short summary
=================
This assertion method checks if the current string ``stringToCheck`` length
is equal to ``expectedLength``

.. <legal notes>

legal notes
=================
| SPDX-FileCopyrightText: © 2022 ekvip automation GmbH <info@ekvip.de>
| SPDX-License-Identifier: Apache-2.0
| For details check: Apache-2.0_

.. _Apache-2.0: https://www.apache.org/licenses/LICENSE-2.0

.. </legal notes>

parameters
=================

*)

METHOD lenghtIsExact
VAR_INPUT
	(* current string to check *)
	stringToCheck	:WSTRING(Tc2_System.MAX_STRING_LENGTH);
	(* expected length of ``stringToCheck`` *)
	expectedLength	:USINT;
	(* message if the assertion is false *)
	message			:AssertMessage;
END_VAR
END_METHOD

(*

short summary
=================
This assertion method checks if the current string ``stringToCheck`` length
is equal or less than to ``maxLength``

.. <legal notes>

legal notes
=================
| SPDX-FileCopyrightText: © 2022 ekvip automation GmbH <info@ekvip.de>
| SPDX-License-Identifier: Apache-2.0
| For details check: Apache-2.0_

.. _Apache-2.0: https://www.apache.org/licenses/LICENSE-2.0

.. </legal notes>

parameters
=================

*)

METHOD lenghtIsMax
VAR_INPUT
	(* current string to check *)
	stringToCheck	:WSTRING(Tc2_System.MAX_STRING_LENGTH);
	(* upper limit of the length of ``stringToCheck`` *)
	maxLength		:USINT;
	(* message if the assertion is false *)
	message			:AssertMessage;
END_VAR
END_METHOD

(*

short summary
=================
This assertion method checks if the current string ``stringToCheck`` length
is equal or grater than to ``minLength``

.. <legal notes>

legal notes
=================
| SPDX-FileCopyrightText: © 2022 ekvip automation GmbH <info@ekvip.de>
| SPDX-License-Identifier: Apache-2.0
| For details check: Apache-2.0_

.. _Apache-2.0: https://www.apache.org/licenses/LICENSE-2.0

.. </legal notes>

parameters
=================

*)

METHOD lenghtIsMin
VAR_INPUT
	(* current string to check *)
	stringToCheck	:WSTRING(Tc2_System.MAX_STRING_LENGTH);
	(* lower limit of the length of ``stringToCheck`` *)
	minLength	:USINT;
	(* message if the assertion is false *)
	message			:AssertMessage;
END_VAR
END_METHOD

(*

short summary
=================
This assertion method checks if the current string ``stringToCheck`` starts with ``start``

.. attention:: 
	start of the string is **ALWAYS** the left side of the string 
	even for writings which written from right to left like Hebrew or Arabic

.. <legal notes>

legal notes
=================
| SPDX-FileCopyrightText: © 2022 ekvip automation GmbH <info@ekvip.de>
| SPDX-License-Identifier: Apache-2.0
| For details check: Apache-2.0_

.. _Apache-2.0: https://www.apache.org/licenses/LICENSE-2.0

.. </legal notes>

parameters
=================

*)

METHOD startsWith
VAR_INPUT
	(* current string to check *)
	stringToCheck	:WSTRING(Tc2_System.MAX_STRING_LENGTH);
	(* expected start of ``stringToCheck`` *)
	start			:WSTRING(Tc2_System.MAX_STRING_LENGTH);
	(* ``TRUE`` means ignore cases; ``FALSE`` means cases must be equal too *)
	ignoreCases		:BOOL;
	(* ``TRUE`` means truncation of spaces on the left side of ``stringToCheck``*)
	trim			:BOOL;
	(* message if the assertion is false *)
	message			:AssertMessage;
END_VAR
END_METHOD

END_INTERFACE

// ---- Assertor/Assertions/StringAssertion/WString/interfaces/IUtf16StringPointerAssertions.TcIO
(*

short summary
=================
This interface provides assert statements for UTF-16 strings

.. attention:: 
	All strings are handled as null terminated word streams.
	For UTF-16 is end of the string 16#00_00

.. <legal notes>

legal notes
=================
| SPDX-FileCopyrightText: © 2022 ekvip automation GmbH <info@ekvip.de>
| SPDX-License-Identifier: Apache-2.0
| For details check: Apache-2.0_

.. _Apache-2.0: https://www.apache.org/licenses/LICENSE-2.0

.. </legal notes>

methods
==================

*)

INTERFACE IUtf16StringPointerAssertions EXTENDS IAssertCallBackSetter

(*

short summary
=================
This assertion method for UTF-16 strings checks if the current string ``stringToCheck`` contains the search string ``searchString``

.. attention:: 
	All strings are handled as null terminated word streams.
	For UTF-16 is end of the string 16#00_00

.. <legal notes>

legal notes
=================
| SPDX-FileCopyrightText: © 2022 ekvip automation GmbH <info@ekvip.de>
| SPDX-License-Identifier: Apache-2.0
| For details check: Apache-2.0_

.. _Apache-2.0: https://www.apache.org/licenses/LICENSE-2.0

.. </legal notes>

parameters
=================

*)

METHOD utf16Contains
VAR_INPUT
	(* current string to check *)
	stringToCheck	:POINTER TO WORD;
	(* string must be found in ``stringToCheck`` *)
	searchString	:POINTER TO WORD;
	(* ``TRUE`` means ignore cases; ``FALSE`` means cases must be equal too *)
	ignoreCases		:BOOL;
	(* message if the assertion is false *)
	message			:AssertMessage;
END_VAR
END_METHOD

(*

short summary
=================
This assertion method for UTF-16 strings checks if the current string ``stringToCheck`` contains not the search string ``searchString``

.. attention:: 
	All strings are handled as null terminated word streams.
	For UTF-16 is end of the string 16#00_00

.. <legal notes>

legal notes
=================
| SPDX-FileCopyrightText: © 2022 ekvip automation GmbH <info@ekvip.de>
| SPDX-License-Identifier: Apache-2.0
| For details check: Apache-2.0_

.. _Apache-2.0: https://www.apache.org/licenses/LICENSE-2.0

.. </legal notes>

parameters
=================

*)

METHOD utf16ContainsNo
VAR_INPUT
	(* current string to check *)
	stringToCheck	:POINTER TO WORD;
	(* string must be found in ``stringToCheck`` *)
	searchString	:POINTER TO WORD;
	(* ``TRUE`` means ignore cases; ``FALSE`` means cases must be equal too *)
	ignoreCases		:BOOL;
	(* message if the assertion is false *)
	message			:AssertMessage;
END_VAR
END_METHOD

(*

short summary
=================
This assertion method for UTF-16 strings checks if the current string ``stringToCheck`` ends with the string ``end``

.. attention:: 
	All strings are handled as null terminated word streams.
	For UTF-16 is end of the string 16#00_00

.. attention:: 
	end of the string is **ALWAYS** the right side of the string 
	even for writings which written from right to left like Hebrew or Arabic

.. <legal notes>

legal notes
=================
| SPDX-FileCopyrightText: © 2022 ekvip automation GmbH <info@ekvip.de>
| SPDX-License-Identifier: Apache-2.0
| For details check: Apache-2.0_

.. _Apache-2.0: https://www.apache.org/licenses/LICENSE-2.0

.. </legal notes>

parameters
=================

*)

METHOD utf16EndsWith
VAR_INPUT
	(* current string to check *)
	stringToCheck	:POINTER TO WORD;
	(* string must be the end of ``stringToCheck`` *)
	end				:POINTER TO WORD;
	(* ``TRUE`` means ignore cases; ``FALSE`` means cases must be equal too *)
	ignoreCases		:BOOL;
	(* ``TRUE`` means truncation of spaces on the right side of ``stringToCheck``*)
	trim			:BOOL;
	(* message if the assertion is false *)
	message			:AssertMessage;
END_VAR
END_METHOD

(*

short summary
=================
This assertion method for utf-16 strings checks if the current string ``stringToCheck`` is equal to the ``expected`` string

.. attention:: 
	All strings are handled as null terminated word streams.
	For UTF-16 is end of the string 16#00_00

.. <legal notes>

legal notes
=================
| SPDX-FileCopyrightText: © 2022 ekvip automation GmbH <info@ekvip.de>
| SPDX-License-Identifier: Apache-2.0
| For details check: Apache-2.0_

.. _Apache-2.0: https://www.apache.org/licenses/LICENSE-2.0

.. </legal notes>

parameters
=================

*)

METHOD utf16IsEqualTo
VAR_INPUT
	(* current string to check *)
	stringToCheck	:POINTER TO WORD;
	(* ``stringToCheck`` must be equal to expected *)
	expected		:POINTER TO WORD;
	(* ``TRUE`` means ignore cases; ``FALSE`` means cases must be equal too *)
	ignoreCases		:BOOL;
	(* message if the assertion is false *)
	message			:AssertMessage;
END_VAR
END_METHOD

(*

short summary
=================
This assertion method for utf-16 strings checks if the current string ``stringToCheck`` is not equal to the ``unexpected`` string

.. attention:: 
	All strings are handled as null terminated word streams.
	For UTF-16 is end of the string 16#00_00

.. <legal notes>

legal notes
=================
| SPDX-FileCopyrightText: © 2022 ekvip automation GmbH <info@ekvip.de>
| SPDX-License-Identifier: Apache-2.0
| For details check: Apache-2.0_

.. _Apache-2.0: https://www.apache.org/licenses/LICENSE-2.0

.. </legal notes>

parameters
=================

*)

METHOD utf16IsNotEqualTo
VAR_INPUT
	(* current string to check *)
	stringToCheck	:POINTER TO WORD;
	(* ``stringToCheck`` must be not equal to unexpected *)
	unexpected		:POINTER TO WORD;
	(* ``TRUE`` means ignore cases; ``FALSE`` means cases must be equal too *)
	ignoreCases		:BOOL;
	(* message if the assertion is false *)
	message			:AssertMessage;
END_VAR
END_METHOD

(*

short summary
=================
This assertion method checks if the current string ``stringToCheck`` is length
is equal to ``expectedLength``

.. attention:: 
	All strings are handled as null terminated word streams.
	For UTF-16 is end of the string 16#00_00

.. <legal notes>

legal notes
=================
| SPDX-FileCopyrightText: © 2022 ekvip automation GmbH <info@ekvip.de>
| SPDX-License-Identifier: Apache-2.0
| For details check: Apache-2.0_

.. _Apache-2.0: https://www.apache.org/licenses/LICENSE-2.0

.. </legal notes>

parameters
=================

*)

METHOD utf16LenghtIsExact
VAR_INPUT
	(* current string to check *)
	stringToCheck	:POINTER TO WORD;
	(* expected length of ``stringToCheck`` *)
	expectedLength	:UDINT;
	(* message if the assertion is false *)
	message			:AssertMessage;
END_VAR
END_METHOD

(*

short summary
=================
This assertion method checks if the current string ``stringToCheck`` is length
is equal or less than to ``maxLength``

.. attention:: 
	All strings are handled as null terminated word streams.
	For UTF-16 is end of the string 16#00_00

.. <legal notes>

legal notes
=================
| SPDX-FileCopyrightText: © 2022 ekvip automation GmbH <info@ekvip.de>
| SPDX-License-Identifier: Apache-2.0
| For details check: Apache-2.0_

.. _Apache-2.0: https://www.apache.org/licenses/LICENSE-2.0

.. </legal notes>

parameters
=================

*)

METHOD utf16LenghtIsMax
VAR_INPUT
	(* current string to check *)
	stringToCheck	:POINTER TO WORD;
	(* upper limit of the length of ``stringToCheck`` *)
	maxLength		:UDINT;
	(* message if the assertion is false *)
	message			:AssertMessage;
END_VAR
END_METHOD

(*

short summary
=================
This assertion method checks if the current string ``stringToCheck`` is length
is equal or grater than to ``minLength``

.. attention:: 
	All strings are handled as null terminated word streams.
	For UTF-16 is end of the string 16#00_00

.. <legal notes>

legal notes
=================
| SPDX-FileCopyrightText: © 2022 ekvip automation GmbH <info@ekvip.de>
| SPDX-License-Identifier: Apache-2.0
| For details check: Apache-2.0_

.. _Apache-2.0: https://www.apache.org/licenses/LICENSE-2.0

.. </legal notes>

parameters
=================

*)

METHOD utf16LenghtIsMin
VAR_INPUT
	(* current string to check *)
	stringToCheck	:POINTER TO WORD;
	(* lower limit of the length of ``stringToCheck`` *)
	minLength		:UDINT;
	(* message if the assertion is false *)
	message			:AssertMessage;
END_VAR
END_METHOD

(*

short summary
=================
This assertion method checks if the current string ``stringToCheck`` is length
is equal or grater than ``minLength`` and equal or less than ``maxLength``

.. attention:: 
	All strings are handled as null terminated word streams.
	For UTF-16 is end of the string 16#00_00

.. <legal notes>

legal notes
=================
| SPDX-FileCopyrightText: © 2022 ekvip automation GmbH <info@ekvip.de>
| SPDX-License-Identifier: Apache-2.0
| For details check: Apache-2.0_

.. _Apache-2.0: https://www.apache.org/licenses/LICENSE-2.0

.. </legal notes>

parameters
=================

*)

METHOD utf16LengthIsBetween
VAR_INPUT
	(* current string to check *)
	stringToCheck	:POINTER TO WORD;
	(* lower limit of the string length *)
	minLenght		:UDINT;
	(* upper limit of the string length *)
	maxLenght		:UDINT;
	(* message if the assertion is false *)
	message			:AssertMessage;
END_VAR
END_METHOD

(*

short summary
=================
This assertion method for UTF-16 strings checks if the current string ``stringToCheck`` strats with the string ``start``

.. attention:: 
	All strings are handled as null terminated word streams.
	For UTF-16 is end of the string 16#00_00

.. attention:: 
	start of the string is **ALWAYS** the left side of the string 
	even for writings which written from right to left like Hebrew or Arabic

.. <legal notes>

legal notes
=================
| SPDX-FileCopyrightText: © 2022 ekvip automation GmbH <info@ekvip.de>
| SPDX-License-Identifier: Apache-2.0
| For details check: Apache-2.0_

.. _Apache-2.0: https://www.apache.org/licenses/LICENSE-2.0

.. </legal notes>

parameters
=================

*)

METHOD utf16StartsWith
VAR_INPUT
	(* current string to check *)
	stringToCheck	:POINTER TO WORD;
	(* expected start of ``stringToCheck`` *)
	start			:POINTER TO WORD;
	(* ``TRUE`` means ignore cases; ``FALSE`` means cases must be equal too *)
	ignoreCases		:BOOL;
	(* ``TRUE`` means truncation of spaces on the right side of ``stringToCheck``*)
	trim			:BOOL;
	(* message if the assertion is false *)
	message			:AssertMessage;
END_VAR
END_METHOD

END_INTERFACE

// ---- Assertor/Assertions/TimeAssertions/interfaces/ITimeAssertions.TcIO
(*

short summary
=================
This interface provides assert statements for times
For ``LTIME`` assertions use the property :ref:`ITimeAssertions.long`.
For ``TIME`` assertions use the property :ref:`ITimeAssertions.simple`.
.. <legal notes>

legal notes
=================
| SPDX-FileCopyrightText: © 2022 ekvip automation GmbH <info@ekvip.de>
| SPDX-License-Identifier: Apache-2.0
| For details check: Apache-2.0_

.. _Apache-2.0: https://www.apache.org/licenses/LICENSE-2.0

.. </legal notes>

methods
==================

*)

INTERFACE ITimeAssertions EXTENDS __SYSTEM.IQueryInterface

(*

short summary
=================
Returns an interface with assert statements for 64 bit times 

.. <legal notes>

legal notes
=================
| SPDX-FileCopyrightText: © 2022 ekvip automation GmbH <info@ekvip.de>
| SPDX-License-Identifier: Apache-2.0
| For details check: Apache-2.0_

.. _Apache-2.0: https://www.apache.org/licenses/LICENSE-2.0

.. </legal notes>

*)

PROPERTY long :I64BitTimeAssertions
GET
END_GET
END_PROPERTY

(*

short summary
=================
Returns an interface with assert statements for 32 bit times 

.. <legal notes>

legal notes
=================
| SPDX-FileCopyrightText: © 2022 ekvip automation GmbH <info@ekvip.de>
| SPDX-License-Identifier: Apache-2.0
| For details check: Apache-2.0_

.. _Apache-2.0: https://www.apache.org/licenses/LICENSE-2.0

.. </legal notes>

*)

PROPERTY simple :I32BitTimeAssertions
GET
END_GET
END_PROPERTY

END_INTERFACE

// ---- Assertor/Assertions/TimeAssertions/LTime/interfaces/I64BitTimeAssertions.TcIO
(*

short summary
=================
This interface provides assert statements for 64 bit ``LTIME``  

.. <legal notes>

legal notes
=================
| SPDX-FileCopyrightText: © 2022 ekvip automation GmbH <info@ekvip.de>
| SPDX-License-Identifier: Apache-2.0
| For details check: Apache-2.0_

.. _Apache-2.0: https://www.apache.org/licenses/LICENSE-2.0

.. </legal notes>

methods
==================

*)

INTERFACE I64BitTimeAssertions EXTENDS __SYSTEM.IQueryInterface

(*

short summary
=================
This assertion method checks whether time has elapsed since the timestamp time

.. <legal notes>

legal notes
=================
| SPDX-FileCopyrightText: © 2022 ekvip automation GmbH <info@ekvip.de>
| SPDX-License-Identifier: Apache-2.0
| For details check: Apache-2.0_

.. _Apache-2.0: https://www.apache.org/licenses/LICENSE-2.0

.. </legal notes>

parameters
=================

*)

METHOD timeHasExpired
VAR_INPUT
	(* start time you get it with ``LTIME()`` *)
	timestamp		:LTIME;
	(* timeout like ``LTIME#300ms`` *)
	expiringTime	:LTIME;
	(* message if the assertion is false *)
	message			:AssertMessage;
END_VAR
END_METHOD

(*

short summary
=================
This assertion method checks that the time since the timestamp time has not yet elapsed

.. <legal notes>

legal notes
=================
| SPDX-FileCopyrightText: © 2022 ekvip automation GmbH <info@ekvip.de>
| SPDX-License-Identifier: Apache-2.0
| For details check: Apache-2.0_

.. _Apache-2.0: https://www.apache.org/licenses/LICENSE-2.0

.. </legal notes>

parameters
=================

*)

METHOD timeHasNotExpired
VAR_INPUT
	(* start time you get it with ``LTIME()`` *)
	timestamp		:LTIME;
	(* timeout like ``LTIME#300ms`` *)
	expiringTime	:LTIME;
	(* message if the assertion is false *)
	message			:AssertMessage;
END_VAR
END_METHOD

(*

short summary
=================
This assertion method checks if the current value is equal to the expected value

.. <legal notes>

legal notes
=================
| SPDX-FileCopyrightText: © 2022 ekvip automation GmbH <info@ekvip.de>
| SPDX-License-Identifier: Apache-2.0
| For details check: Apache-2.0_

.. _Apache-2.0: https://www.apache.org/licenses/LICENSE-2.0

.. </legal notes>

parameters
=================

*)

METHOD valueIsEqualTo
VAR_INPUT
	(* current value to check *)
	currentValue	:LTIME;
	(* expected value to compare *)
	expectedValue	:LTIME;
	(* message if the assertion is false *)
	message			:AssertMessage;
END_VAR
END_METHOD

(*

short summary
=================
This assertion method checks if the current value is greater than the less value

.. <legal notes>

legal notes
=================
| SPDX-FileCopyrightText: © 2022 ekvip automation GmbH <info@ekvip.de>
| SPDX-License-Identifier: Apache-2.0
| For details check: Apache-2.0_

.. _Apache-2.0: https://www.apache.org/licenses/LICENSE-2.0

.. </legal notes>

parameters
=================

*)

METHOD valueIsGreaterThan
VAR_INPUT
	(* current value to check *)
	currentValue	:LTIME;
	(* less than lower limit *)
	lessValue		:LTIME;
	(* message if the assertion is false *)
	message			:AssertMessage;
END_VAR
END_METHOD

(*

short summary
=================
This assertion method checks if the current value is inside a limit

.. attention:: 
	limits are included: ``valueIsInRangeOf(lt#3ms,lt#3ms ,lt#3ms)`` is a true assertion

.. <legal notes>

legal notes
=================
| SPDX-FileCopyrightText: © 2022 ekvip automation GmbH <info@ekvip.de>
| SPDX-License-Identifier: Apache-2.0
| For details check: Apache-2.0_

.. _Apache-2.0: https://www.apache.org/licenses/LICENSE-2.0

.. </legal notes>

parameters
=================

*)

METHOD valueIsInRangeOf
VAR_INPUT
	(* lower limit for the current value *)
	lowerLimit		:LTIME;
	(* current value to check *)
	currentValue	:LTIME;
	(* upper limit for the current value *)
	upperLimit		:LTIME;
	(* message if the assertion is false *)
	message			:AssertMessage;
END_VAR
END_METHOD

(*

short summary
=================
This assertion method checks if the current value is less than the greater value

.. <legal notes>

legal notes
=================
| SPDX-FileCopyrightText: © 2022 ekvip automation GmbH <info@ekvip.de>
| SPDX-License-Identifier: Apache-2.0
| For details check: Apache-2.0_

.. _Apache-2.0: https://www.apache.org/licenses/LICENSE-2.0

.. </legal notes>

parameters
=================

*)

METHOD valueIsLessThan
VAR_INPUT
	(* current value to check *)
	currentValue	:LTIME;
	(* greater than upper limit *)
	greaterValue	:LTIME;
	(* message if the assertion is false *)
	message			:AssertMessage;
END_VAR
END_METHOD

(*

short summary
=================
This assertion method checks if the current value is less than or equal to the maximum value

.. <legal notes>

legal notes
=================
| SPDX-FileCopyrightText: © 2022 ekvip automation GmbH <info@ekvip.de>
| SPDX-License-Identifier: Apache-2.0
| For details check: Apache-2.0_

.. _Apache-2.0: https://www.apache.org/licenses/LICENSE-2.0

.. </legal notes>

parameters
=================

*)

METHOD valueIsMax
VAR_INPUT
	(* current value to check *)
	currentValue	:LTIME;
	(* upper limit for the current value *)
	maximumValue	:LTIME;
	(* message if the assertion is false *)
	message			:AssertMessage;
END_VAR
END_METHOD

(*

short summary
=================
This assertion method checks if the current value is greater than or equal to the minimum value

.. <legal notes>

legal notes
=================
| SPDX-FileCopyrightText: © 2022 ekvip automation GmbH <info@ekvip.de>
| SPDX-License-Identifier: Apache-2.0
| For details check: Apache-2.0_

.. _Apache-2.0: https://www.apache.org/licenses/LICENSE-2.0

.. </legal notes>

parameters
=================

*)

METHOD valueIsMin
VAR_INPUT
	(* current value to check *)
	currentValue	:LTIME;
	(* lower limit for the current value *)
	minimumValue	:LTIME;
	(* message if the assertion is false *)
	message			:AssertMessage;
END_VAR
END_METHOD

(*

short summary
=================
This assertion method checks if the current value is not equal to the unexpected value

.. <legal notes>

legal notes
=================
| SPDX-FileCopyrightText: © 2022 ekvip automation GmbH <info@ekvip.de>
| SPDX-License-Identifier: Apache-2.0
| For details check: Apache-2.0_

.. _Apache-2.0: https://www.apache.org/licenses/LICENSE-2.0

.. </legal notes>

parameters
=================

*)

METHOD valueIsNotEqualTo
VAR_INPUT
	(* current value to check *)
	currentValue	:LTIME;
	(* unexpected value to compare *)
	unexpectedValue	:LTIME;
	(* message if the assertion is false *)
	message			:AssertMessage;
END_VAR
END_METHOD

END_INTERFACE

// ---- Assertor/Assertions/TimeAssertions/Time/interfaces/I32BitTimeAssertions.TcIO
(*

short summary
=================
This interface provides assert statements for 32 bit ``TIME``  

.. <legal notes>

legal notes
=================
| SPDX-FileCopyrightText: © 2022 ekvip automation GmbH <info@ekvip.de>
| SPDX-License-Identifier: Apache-2.0
| For details check: Apache-2.0_

.. _Apache-2.0: https://www.apache.org/licenses/LICENSE-2.0

.. </legal notes>

methods
==================

*)

INTERFACE I32BitTimeAssertions EXTENDS __SYSTEM.IQueryInterface

(*

short summary
=================
This assertion method checks whether time has elapsed since the timestamp time

.. <legal notes>

legal notes
=================
| SPDX-FileCopyrightText: © 2022 ekvip automation GmbH <info@ekvip.de>
| SPDX-License-Identifier: Apache-2.0
| For details check: Apache-2.0_

.. _Apache-2.0: https://www.apache.org/licenses/LICENSE-2.0

.. </legal notes>

parameters
=================

*)

METHOD timeHasExpired
VAR_INPUT
	(* start time you get it with ``TIME()`` *)
	timestamp		:TIME;
	(* timeout like ``t#300ms`` *)
	expiringTime	:TIME;
	(* message if the assertion is false *)
	message			:AssertMessage;
END_VAR
END_METHOD

(*

short summary
=================
This assertion method checks that the time since the timestamp time has not yet elapsed

.. <legal notes>

legal notes
=================
| SPDX-FileCopyrightText: © 2022 ekvip automation GmbH <info@ekvip.de>
| SPDX-License-Identifier: Apache-2.0
| For details check: Apache-2.0_

.. _Apache-2.0: https://www.apache.org/licenses/LICENSE-2.0

.. </legal notes>

parameters
=================

*)

METHOD timeHasNotExpired
VAR_INPUT
	(* start time you get it with ``TIME()`` *)
	timestamp		:TIME;
	(* timeout like ``t#300ms`` *)
	expiringTime	:TIME;
	(* message if the assertion is false *)
	message			:AssertMessage;
END_VAR
END_METHOD

(*

short summary
=================
This assertion method checks if the current value is equal to the expected value

.. <legal notes>

legal notes
=================
| SPDX-FileCopyrightText: © 2022 ekvip automation GmbH <info@ekvip.de>
| SPDX-License-Identifier: Apache-2.0
| For details check: Apache-2.0_

.. _Apache-2.0: https://www.apache.org/licenses/LICENSE-2.0

.. </legal notes>

parameters
=================

*)

METHOD valueIsEqualTo
VAR_INPUT
	(* current value to check *)
	currentValue	:TIME;
	(* expected value to compare *)
	expectedValue	:TIME;
	(* message if the assertion is false *)
	message			:AssertMessage;
END_VAR
END_METHOD

(*

short summary
=================
This assertion method checks if the current value is greater than the less value

.. <legal notes>

legal notes
=================
| SPDX-FileCopyrightText: © 2022 ekvip automation GmbH <info@ekvip.de>
| SPDX-License-Identifier: Apache-2.0
| For details check: Apache-2.0_

.. _Apache-2.0: https://www.apache.org/licenses/LICENSE-2.0

.. </legal notes>

parameters
=================

*)

METHOD valueIsGreaterThan
VAR_INPUT
	(* current value to check *)
	currentValue	:TIME;
	(* less than lower limit *)
	lessValue		:TIME;
	(* message if the assertion is false *)
	message			:AssertMessage;
END_VAR
END_METHOD

(*

short summary
=================
This assertion method checks if the current value is inside a limit

.. attention:: 
	limits are included: ``valueIsInRangeOf(t#3ms,t#3ms ,t#3ms)`` is a true assertion

.. <legal notes>

legal notes
=================
| SPDX-FileCopyrightText: © 2022 ekvip automation GmbH <info@ekvip.de>
| SPDX-License-Identifier: Apache-2.0
| For details check: Apache-2.0_

.. _Apache-2.0: https://www.apache.org/licenses/LICENSE-2.0

.. </legal notes>

parameters
=================

*)

METHOD valueIsInRangeOf
VAR_INPUT
	(* lower limit for the current value *)
	lowerLimit		:TIME;
	(* current value to check *)
	currentValue	:TIME;
	(* upper limit for the current value *)
	upperLimit		:TIME;
	(* message if the assertion is false *)
	message			:AssertMessage;
END_VAR
END_METHOD

(*

short summary
=================
This assertion method checks if the current value is less than the greater value

.. <legal notes>

legal notes
=================
| SPDX-FileCopyrightText: © 2022 ekvip automation GmbH <info@ekvip.de>
| SPDX-License-Identifier: Apache-2.0
| For details check: Apache-2.0_

.. _Apache-2.0: https://www.apache.org/licenses/LICENSE-2.0

.. </legal notes>

parameters
=================

*)

METHOD valueIsLessThan
VAR_INPUT
	(* current value to check *)
	currentValue	:TIME;
	(* greater than upper limit *)
	greaterValue	:TIME;
	(* message if the assertion is false *)
	message			:AssertMessage;
END_VAR
END_METHOD

(*

short summary
=================
This assertion method checks if the current value is less than or equal to the maximum value

.. <legal notes>

legal notes
=================
| SPDX-FileCopyrightText: © 2022 ekvip automation GmbH <info@ekvip.de>
| SPDX-License-Identifier: Apache-2.0
| For details check: Apache-2.0_

.. _Apache-2.0: https://www.apache.org/licenses/LICENSE-2.0

.. </legal notes>

parameters
=================

*)

METHOD valueIsMax
VAR_INPUT
	(* current value to check *)
	currentValue	:TIME;
	(* upper limit for the current value *)
	maximumValue	:TIME;
	(* message if the assertion is false *)
	message			:AssertMessage;
END_VAR
END_METHOD

(*

short summary
=================
This assertion method checks if the current value is greater than or equal to the minimum value

.. <legal notes>

legal notes
=================
| SPDX-FileCopyrightText: © 2022 ekvip automation GmbH <info@ekvip.de>
| SPDX-License-Identifier: Apache-2.0
| For details check: Apache-2.0_

.. _Apache-2.0: https://www.apache.org/licenses/LICENSE-2.0

.. </legal notes>

parameters
=================

*)

METHOD valueIsMin
VAR_INPUT
	(* current value to check *)
	currentValue	:TIME;
	(* lower limit for the current value *)
	minimumValue	:TIME;
	(* message if the assertion is false *)
	message			:AssertMessage;
END_VAR
END_METHOD

(*

short summary
=================
This assertion method checks if the current value is not equal to the unexpected value

.. <legal notes>

legal notes
=================
| SPDX-FileCopyrightText: © 2022 ekvip automation GmbH <info@ekvip.de>
| SPDX-License-Identifier: Apache-2.0
| For details check: Apache-2.0_

.. _Apache-2.0: https://www.apache.org/licenses/LICENSE-2.0

.. </legal notes>

parameters
=================

*)

METHOD valueIsNotEqualTo
VAR_INPUT
	(* current value to check *)
	currentValue	:TIME;
	(* unexpected value to compare *)
	unexpectedValue	:TIME;
	(* message if the assertion is false *)
	message			:AssertMessage;
END_VAR
END_METHOD

END_INTERFACE

// ---- Assertor/interfaces/IAssertor.TcIO
(*

short summary
=================
This interface provides assert statements
for the most common data types. The interface
is made to avoid to many methods to select in 
intelliSense of the TwinCAT editor

.. <legal notes>

legal notes
=================
| SPDX-FileCopyrightText: © 2022 ekvip automation GmbH <info@ekvip.de>
| SPDX-License-Identifier: Apache-2.0
| For details check: Apache-2.0_

.. _Apache-2.0: https://www.apache.org/licenses/LICENSE-2.0

.. </legal notes>

properties
==================

*)

INTERFACE IAssertor EXTENDS __SYSTEM.IQueryInterface

(*

short summary
=================
Returns the interface :ref:`IAssertions`
to get access to the assert statements

.. <legal notes>

legal notes
=================
| SPDX-FileCopyrightText: © 2022 ekvip automation GmbH <info@ekvip.de>
| SPDX-License-Identifier: Apache-2.0
| For details check: Apache-2.0_

.. _Apache-2.0: https://www.apache.org/licenses/LICENSE-2.0

.. </legal notes>

methods
==================

*)

PROPERTY assert :IAssertions
GET
END_GET
END_PROPERTY

END_INTERFACE

// ---- Assertor/interfaces/IAssertCallBack.TcIO
(*

short summary
=================
This interface provides the a callback
method for which is called if an assertions
is worng

.. <legal notes>

legal notes
=================
| SPDX-FileCopyrightText: © 2022 ekvip automation GmbH <info@ekvip.de>
| SPDX-License-Identifier: Apache-2.0
| For details check: Apache-2.0_

.. _Apache-2.0: https://www.apache.org/licenses/LICENSE-2.0

.. </legal notes>

methods
==================

*)

INTERFACE IAssertCallBack EXTENDS CNM_AbstractObject.IObject

(*

short summary
=================
This method is called if an assertion was ``FALSE``

.. <legal notes>

legal notes
=================
| SPDX-FileCopyrightText: © 2022 ekvip automation GmbH <info@ekvip.de>
| SPDX-License-Identifier: Apache-2.0
| For details check: Apache-2.0_

.. _Apache-2.0: https://www.apache.org/licenses/LICENSE-2.0

.. </legal notes>

parameters
=================

*)

METHOD assertionWasWrong
VAR_INPUT
	(* caller object of the method *)
	caller			:CNM_AbstractObject.IObject;
	(* alarm message *)
	message			:AssertMessage;
	(* debugging information *) 
	additionalText	:Tc2_System.T_MaxString;
END_VAR
END_METHOD

END_INTERFACE

// ---- Assertor/interfaces/IAssertCallBackSetter.TcIO
(*

short summary
=================
This interface provides the possibilty to set a callback class 

.. <legal notes>

legal notes
=================
| SPDX-FileCopyrightText: © 2022 ekvip automation GmbH <info@ekvip.de>
| SPDX-License-Identifier: Apache-2.0
| For details check: Apache-2.0_

.. _Apache-2.0: https://www.apache.org/licenses/LICENSE-2.0

.. </legal notes>

methods
==================

*)

INTERFACE IAssertCallBackSetter EXTENDS CNM_AbstractObject.IObject

(*

short summary
=================
This methods is the setter for the callback class if an assertion was false

.. <legal notes>

legal notes
=================
| SPDX-FileCopyrightText: © 2022 ekvip automation GmbH <info@ekvip.de>
| SPDX-License-Identifier: Apache-2.0
| For details check: Apache-2.0_

.. _Apache-2.0: https://www.apache.org/licenses/LICENSE-2.0

.. </legal notes>

parameters
=================

*)

METHOD setCallBack
VAR_INPUT
	(* the class that must be informed if an assertion is false *)
	callBack	:IAssertCallback;  
END_VAR
END_METHOD

END_INTERFACE

// ---- Assertor/Assertions/BinaryAssertions/classes/BinaryAssertions.TcPOU
(*

short summary
=================
This class provides assert statements for binaries
e.g. structures, arrays etc...
It implements the interface :ref:`IBinaryAssertions`

.. <legal notes>

legal notes
=================
| SPDX-FileCopyrightText: © 2022 ekvip automation GmbH <info@ekvip.de>
| SPDX-License-Identifier: Apache-2.0
| For details check: Apache-2.0_

.. _Apache-2.0: https://www.apache.org/licenses/LICENSE-2.0

.. </legal notes>

methods and properties
=======================

*)

{attribute 'reflection'}
FUNCTION_BLOCK INTERNAL BinaryAssertions EXTENDS AbstactAssertion IMPLEMENTS IBinaryAssertions
VAR CONSTANT
	(* to check if binary data points to nowhere *)
	NULL_POINTER	:POINTER TO BYTE := 0;
	(* to check if the binary data has no size *)
	ZERO_SIZE		:DINT := 0;
	(* register size of the plattform, shall be always 8 byte *)
	REGISTER_SIZE	:DINT := SIZEOF(__XWORD);
	(* first index of a pointer *) 
	FIRST_DATA		:LINT := 0;
	(* direction for little endian *)
	DIRECTION_LE	:LINT := -1;
END_VAR

(*

short summary
=================
This method comapres the data of two any pointers. 
The table below shows with some examples how it works.

+-------------------+------------------+----------------------------+---------------------------+---------------------------------------+
| **value of data** | **size of data** | **value of dataToCompare** | **size of dataToCompare** | **CNM_ReturnTypes.ComparationResult** |
+===================+==================+============================+===========================+=======================================+
| null              | 0                | null                       | 0                         | EQUAL                                 |
+-------------------+------------------+----------------------------+---------------------------+---------------------------------------+
| null              | 0                | 16#01                      | 1                         | SMALLER                               |
+-------------------+------------------+----------------------------+---------------------------+---------------------------------------+
| 16#01             | 1                | null                       | 0                         | GREATER                               |
+-------------------+------------------+----------------------------+---------------------------+---------------------------------------+
| 16#00FF           | 2                | 16#FF                      | 1                         | EQUAL                                 |
+-------------------+------------------+----------------------------+---------------------------+---------------------------------------+
| 16#0100           | 2                | 16#FF                      | 1                         | GREATER                               |
+-------------------+------------------+----------------------------+---------------------------+---------------------------------------+
| 16#FF             | 1                | 16#0100                    | 2                         | SMALLER                               |
+-------------------+------------------+----------------------------+---------------------------+---------------------------------------+
| 16#FF             | 1                | 16#00FF                    | 2                         | EQUAL                                 |
+-------------------+------------------+----------------------------+---------------------------+---------------------------------------+
| 16#0FF0           | 2                | 16#F00F                    | 2                         | SMALLER                               |
+-------------------+------------------+----------------------------+---------------------------+---------------------------------------+

.. attention:: 
	Binary comparison means it compares values byte by byte, regardless of type information (signs, ``REAL`` etc...)
	and it compares padding bytes, too.

.. attention:: 
	``STRING`` and ``WSTRING`` is null terminated
	that means TwinCAT sets null byte/word at the end of the string and touches nothing else
	For example ``foo :STRING(3) := 'foo';`` looks binary 16#66 16#6F 16#6F 16#00.
	if you set foo to an empty string ``foo := ''`` it looks like 16#00 16#6F 16#6F 16#00.

.. attention:: 
	It works not for bits because the minimum size must be at least one byte. If the ``__SYSTEM.TYPE_CLASS``
	of ``data`` ``AND`` ``dataToCompare is ``__SYSTEM.TYPE_CLASS.TYPE_BOOL`` ``OR`` ``__SYSTEM.TYPE_CLASS.TYPE_BIT``
	it uses the ``TO_BOOL`` operator for comarison. That means for ``__SYSTEM.TYPE_CLASS.TYPE_BIT`` it has no idea
	if the single ``BIT`` is set or unset, it compares just the whole ``BYTE``.

.. <legal notes>

legal notes
=================
| SPDX-FileCopyrightText: © 2022 ekvip automation GmbH <info@ekvip.de>
| SPDX-License-Identifier: Apache-2.0
| For details check: Apache-2.0_

.. _Apache-2.0: https://www.apache.org/licenses/LICENSE-2.0

.. </legal notes>

parameters
=================
:return: ``SMALLER``: ``data`` is smaller than ``dataToCompare``, 
``EQUAL``: ``data`` is equal to ``dataToCompare``,
``Greater``: ``data`` is greater to ``dataToCompare``

*)

METHOD PROTECTED binaryCompare :CNM_ReturnTypes.ComparationResult
VAR_INPUT
	(* current binary data *)
	data			:ANY;
	(* binary data with smaller values *)
	dataToCompare	:ANY;
END_VAR
VAR CONSTANT
	(* for boolens to figure out if the size exactly one byte *) 
	SIZE_OF_ONE_BYTE	:DINT := 1;
END_VAR
binaryCompare := CNM_ReturnTypes.ComparationResult.EQUAL;
RETURN ((data.pValue = THIS^.NULL_POINTER) AND (dataToCompare.pValue = THIS^.NULL_POINTER));
RETURN ((data.diSize = THIS^.ZERO_SIZE) AND (dataToCompare.diSize = THIS^.ZERO_SIZE));
IF (
	((data.pValue = THIS^.NULL_POINTER) AND (dataToCompare.pValue <> THIS^.NULL_POINTER))
	OR ((data.diSize = THIS^.ZERO_SIZE) AND (dataToCompare.diSize <> THIS^.ZERO_SIZE))
)THEN
	binaryCompare := CNM_ReturnTypes.ComparationResult.SMALLER;
ELSIF (
	((data.pValue <> THIS^.NULL_POINTER) AND (dataToCompare.pValue = THIS^.NULL_POINTER))
	OR ((data.diSize <> THIS^.ZERO_SIZE) AND (dataToCompare.diSize = THIS^.ZERO_SIZE))
)THEN
	binaryCompare := CNM_ReturnTypes.ComparationResult.GREATER;
ELSIF (data.diSize < dataToCompare.diSize) THEN
	IF (THIS^.isDataZero(
		data := dataToCompare.pValue,
		size := dataToCompare.diSize,
		end := dataToCompare.diSize - data.diSize
	)) THEN
		binaryCompare := THIS^.compareData(
			data := data.pValue,
			dataToCompare := dataToCompare.pValue,
			size := data.diSize
		);
	ELSE
		binaryCompare := CNM_ReturnTypes.ComparationResult.SMALLER;
	END_IF
ELSIF (data.diSize > dataToCompare.diSize) THEN
	IF (THIS^.isDataZero(
		data := data.pValue,
		size := data.diSize,
		end := data.diSize - dataToCompare.diSize
	)) THEN
		binaryCompare := THIS^.compareData(
			data := data.pValue,
			dataToCompare := dataToCompare.pValue,
			size := dataToCompare.diSize
		);
	ELSE
		binaryCompare := CNM_ReturnTypes.ComparationResult.GREATER;
	END_IF
ELSIF (
	(data.diSize = SIZE_OF_ONE_BYTE)
	AND (dataToCompare.diSize = SIZE_OF_ONE_BYTE)
	AND (
		(data.TypeClass = __SYSTEM.TYPE_CLASS.TYPE_BOOL)
		OR (data.TypeClass = __SYSTEM.TYPE_CLASS.TYPE_BIT)
	)AND(
		(dataToCompare.TypeClass = __SYSTEM.TYPE_CLASS.TYPE_BOOL)
		OR (dataToCompare.TypeClass = __SYSTEM.TYPE_CLASS.TYPE_BIT)
	)	
)THEN
	IF (TO_BOOL(data.pValue^) AND (NOT TO_BOOL(dataToCompare.pValue^))) THEN
		binaryCompare := CNM_ReturnTypes.ComparationResult.GREATER;
	ELSIF  ((NOT TO_BOOL(data.pValue^)) AND TO_BOOL(dataToCompare.pValue^)) THEN
		binaryCompare := CNM_ReturnTypes.ComparationResult.SMALLER;
	END_IF
ELSIF (data.diSize = dataToCompare.diSize) THEN
	binaryCompare := THIS^.compareData(
		data := data.pValue,
		dataToCompare := dataToCompare.pValue,
		size := data.diSize
	);
END_IF
END_METHOD

(*

short summary
=================
This abstract property returns the class name of the concrete object, 
It's for debugging purpose

.. <legal notes>

legal notes
=================
| SPDX-FileCopyrightText: © 2022 ekvip automation GmbH <info@ekvip.de>
| SPDX-License-Identifier: Apache-2.0
| For details check: Apache-2.0_

.. _Apache-2.0: https://www.apache.org/licenses/LICENSE-2.0

.. </legal notes>

*)

PROPERTY className :CNM_AbstractObject.ClassName
GET
className := 'CNM_AssertionInterfaceLib.BinaryAssertions';
END_GET
END_PROPERTY

(*

short summary
=================
This method comapres the data of two byte pointers. 
The table below shows with some examples how it works.

+-------------------+----------------------------+----------+---------------------------------------+
| **value of data** | **value of dataToCompare** | **size** | **CNM_ReturnTypes.ComparationResult** |
+===================+============================+==========+=======================================+
| 16#00FF           | 16#FF                      | 1        | EQUAL                                 |
+-------------------+----------------------------+----------+---------------------------------------+
| 16#0100           | 16#FF                      | 1        | SMALLER                               |
+-------------------+----------------------------+----------+---------------------------------------+
| 16#FF             | 16#0100                    | 1        | GREATER                               |
+-------------------+----------------------------+----------+---------------------------------------+
| 16#FF             | 16#00FF                    | 1        | EQUAL                                 |
+-------------------+----------------------------+----------+---------------------------------------+
| 16#0FF0           | 16#F00F                    | 1        | GREATER                               |
+-------------------+----------------------------+----------+---------------------------------------+
| 16#0FF0           | 16#F00F                    | 2        | SMALLER                               |
+-------------------+----------------------------+----------+---------------------------------------+

.. attention:: 
	Binary comparison means it compares values byte by byte, regardless of type information (signs, ``REAL`` etc...)
	and it compares padding bytes, too.

.. attention:: 
	``STRING`` and ``WSTRING`` is null terminated
	that means TwinCAT sets null byte/word at the end of the string and touches nothing else
	For example ``foo :STRING(3) := 'foo';`` looks binary 16#66 16#6F 16#6F 16#00.
	if you set foo to an empty string ``foo := ''`` it looks like 16#00 16#6F 16#6F 16#00.

.. <legal notes>

legal notes
=================
| SPDX-FileCopyrightText: © 2022 ekvip automation GmbH <info@ekvip.de>
| SPDX-License-Identifier: Apache-2.0
| For details check: Apache-2.0_

.. _Apache-2.0: https://www.apache.org/licenses/LICENSE-2.0

.. </legal notes>

parameters
=================
:return: ``SMALLER``: ``data`` is smaller than ``dataToCompare``, 
``EQUAL``: ``data`` is equal to ``dataToCompare``,
``Greater``: ``data`` is greater to ``dataToCompare``

*)

METHOD PROTECTED compareBytewise :CNM_ReturnTypes.ComparationResult
VAR_INPUT
	(* current binary data *)
	data			:POINTER TO BYTE;
	(* current binary data to compare *)
	dataToCompare	:POINTER TO BYTE;
	(* size to compare in bytes, it must be smaller or equal to the smaller size of both data *)
	size			:DINT;
	(* last address to comapre *)
	end				:LINT;
END_VAR
VAR
	(* index of the current address *)
	pointerIndex	:LINT;
END_VAR
compareBytewise := CNM_ReturnTypes.ComparationResult.EQUAL;

FOR pointerIndex := (size-1) TO end BY THIS^.DIRECTION_LE DO
	IF (data[pointerIndex] < dataToCompare[pointerIndex]) THEN
		compareBytewise := CNM_ReturnTypes.ComparationResult.SMALLER;
		RETURN;
	ELSIF (data[pointerIndex] > dataToCompare[pointerIndex]) THEN
		compareBytewise := CNM_ReturnTypes.ComparationResult.GREATER;
		RETURN;
	END_IF
END_FOR;
END_METHOD

(*

short summary
=================
This method comapres the data of two byte pointers.
It tries to compare registerwise if it makes sens (pointers are aligned and size big enough)
The table below shows with some examples how it works.

+-------------------+------------------+----------------------------+---------------------------+---------------------------------------+
| **value of data** | **size of data** | **value of dataToCompare** | **size of dataToCompare** | **CNM_ReturnTypes.ComparationResult** |
+===================+==================+============================+===========================+=======================================+
| 16#00FF           | 2                | 16#FF                      | 1                         | EQUAL                                 |
+-------------------+------------------+----------------------------+---------------------------+---------------------------------------+
| 16#0100           | 2                | 16#FF                      | 1                         | GREATER                               |
+-------------------+------------------+----------------------------+---------------------------+---------------------------------------+
| 16#FF             | 1                | 16#0100                    | 2                         | SMALLER                               |
+-------------------+------------------+----------------------------+---------------------------+---------------------------------------+
| 16#FF             | 1                | 16#00FF                    | 2                         | EQUAL                                 |
+-------------------+------------------+----------------------------+---------------------------+---------------------------------------+
| 16#0FF0           | 2                | 16#F00F                    | 2                         | SMALLER                               |
+-------------------+------------------+----------------------------+---------------------------+---------------------------------------+

.. attention:: 
	Binary comparison means it compares values byte by byte, regardless of type information (signs, ``REAL`` etc...)
	and it compares padding bytes, too.

.. attention:: 
	``STRING`` and ``WSTRING`` is null terminated
	that means TwinCAT sets null byte/word at the end of the string and touches nothing else
	For example ``foo :STRING(3) := 'foo';`` looks binary 16#66 16#6F 16#6F 16#00.
	if you set foo to an empty string ``foo := ''`` it looks like 16#00 16#6F 16#6F 16#00.

.. <legal notes>

legal notes
=================
| SPDX-FileCopyrightText: © 2022 ekvip automation GmbH <info@ekvip.de>
| SPDX-License-Identifier: Apache-2.0
| For details check: Apache-2.0_

.. _Apache-2.0: https://www.apache.org/licenses/LICENSE-2.0

.. </legal notes>

parameters
=================
:return: ``SMALLER``: ``data`` is smaller than ``dataToCompare``, 
``EQUAL``: ``data`` is equal to ``dataToCompare``,
``Greater``: ``data`` is greater to ``dataToCompare``

*)

METHOD PROTECTED compareData :CNM_ReturnTypes.ComparationResult
VAR_INPUT
	(* current binary data *)
	data			:POINTER TO BYTE;
	(* current binary data to compare *)
	dataToCompare	:POINTER TO BYTE;
	(* size to compare in bytes, it must be smaller or equal to the smaller size of both data *)
	size			:DINT;
END_VAR
VAR
	(* just a flag to store if both pointer addresses are aligned *)
	arePointersAligned			:BOOL;
	(* number of remaining bytes if it iterates regiterwise through the data*)
	remainingBytes				:DINT;
END_VAR
arePointersAligned := (THIS^.isPointerAligend(data) AND THIS^.isPointerAligend(dataToCompare));

IF (arePointersAligned AND (size >= THIS^.REGISTER_SIZE)) THEN
	remainingBytes := THIS^.getRemainingBytes(size);
	IF (remainingBytes > THIS^.ZERO_SIZE) THEN
		compareData := THIS^.compareBytewise(
			data := data,
			dataToCompare := dataToCompare,
			size := size,
			end := (size - remainingBytes)
		);
		RETURN (compareData <> CNM_ReturnTypes.ComparationResult.EQUAL);
	END_IF
	compareData := THIS^.compareRegisterwise(
		data := data,
		dataToCompare := dataToCompare,
		size := (size - remainingBytes)
	);	
ELSE	
	compareData := THIS^.compareBytewise(
		data := data,
		dataToCompare := dataToCompare,
		size := size,
		end := THIS^.FIRST_DATA
	);
END_IF
END_METHOD

(*

short summary
=================
This method comapres the data of two byte pointers, but it iterates registerwise through the data.
The table below shows with some examples how it works.

+------------------------+----------------------------+----------+---------------------------------------+
|    **value of data**   | **value of dataToCompare** | **size** | **CNM_ReturnTypes.ComparationResult** |
+========================+============================+==========+=======================================+
| 16#00FF_FFFF_0000_FFFF | 16#00FF_FFFF_0000_FFFF     | 8        | EQUAL                                 |
+------------------------+----------------------------+----------+---------------------------------------+
| 16#00FF_FFFF_0000_FFFF | 16#80FF_FFFF_0000_FFFF     | 8        | SMALLER                               |
+------------------------+----------------------------+----------+---------------------------------------+
| 16#80FF_FFFF_0000_FFFF | 16#00FF_FFFF_0000_FFFF     | 8        | GREATER                               |
+------------------------+----------------------------+----------+---------------------------------------+
| 16#FFFF_FFFF_0000_FFFF | 16#FFFF_FFFF_0000_FFFF     | 8        | EQUAL                                 |
+------------------------+----------------------------+----------+---------------------------------------+
| 16#80FF_FFFF_0000_FFFF | 16#70FF_FFFF_FFFF_FFFF     | 8        | GREATER                               |
+------------------------+----------------------------+----------+---------------------------------------+
| 16#70FF_FFFF_FFFF_FFFF | 16#80FF_FFFF_0000_FFFF     | 8        | SMALLER                               |
+------------------------+----------------------------+----------+---------------------------------------+

.. attention:: 
	Binary comparison means it compares values register by register, regardless of type information (signs, ``REAL`` etc...)
	and it compares padding bytes, too.

.. attention:: 
	``STRING`` and ``WSTRING`` is null terminated
	that means TwinCAT sets null byte/word at the end of the string and touches nothing else
	For example ``foo :STRING(3) := 'foo';`` looks binary 16#66 16#6F 16#6F 16#00.
	if you set foo to an empty string ``foo := ''`` it looks like 16#00 16#6F 16#6F 16#00.

.. <legal notes>

legal notes
=================
| SPDX-FileCopyrightText: © 2022 ekvip automation GmbH <info@ekvip.de>
| SPDX-License-Identifier: Apache-2.0
| For details check: Apache-2.0_

.. _Apache-2.0: https://www.apache.org/licenses/LICENSE-2.0

.. </legal notes>

parameters
=================
:return: ``SMALLER``: ``data`` is smaller than ``dataToCompare``, 
``EQUAL``: ``data`` is equal to ``dataToCompare``,
``Greater``: ``data`` is greater to ``dataToCompare``

*)

METHOD PROTECTED compareRegisterwise :CNM_ReturnTypes.ComparationResult
VAR_INPUT
	(* current binary data *)
	data			:POINTER TO __XWORD;
	(* current binary data to compare *)
	dataToCompare	:POINTER TO __XWORD;
	(* size to compare in bytes, size must be a muliple of register size *)
	size			:DINT;
END_VAR
VAR
	(* index of the current address *)
	pointerIndex	:LINT;
END_VAR
VAR CONSTANT
	(* direction for little endian *)
	DIRECTION_LE	:LINT := -1;
END_VAR
compareRegisterwise := CNM_ReturnTypes.ComparationResult.EQUAL;

FOR pointerIndex := (((size)/THIS^.REGISTER_SIZE)-1) TO THIS^.FIRST_DATA BY THIS^.DIRECTION_LE DO
	IF (data[pointerIndex] < dataToCompare[pointerIndex]) THEN
		compareRegisterwise := CNM_ReturnTypes.ComparationResult.SMALLER;
		RETURN;
	ELSIF (data[pointerIndex] > dataToCompare[pointerIndex]) THEN
		compareRegisterwise := CNM_ReturnTypes.ComparationResult.GREATER;
		RETURN;
	END_IF
END_FOR;
END_METHOD

(*

short summary
=================
This method calculates the number of bytes that are remaining
if size is devided by register size.

.. <legal notes>

legal notes
=================
| SPDX-FileCopyrightText: © 2022 ekvip automation GmbH <info@ekvip.de>
| SPDX-License-Identifier: Apache-2.0
| For details check: Apache-2.0_

.. _Apache-2.0: https://www.apache.org/licenses/LICENSE-2.0

.. </legal notes>

parameters
=================
:return: number of bytes that are remaining if it iterates registerwise through the data

*)

METHOD PROTECTED getRemainingBytes :DINT
VAR_INPUT
	(* size in bytes *)
	size			:DINT;
END_VAR
getRemainingBytes := (size MOD THIS^.REGISTER_SIZE);
END_METHOD

(*

short summary
=================
This method checks if the data of a pointer is zero through all bytes (``size-1``)

+------------------------+----------+---------+------------------+
|    **value of data**   | **size** | **end** | **return value** |
+========================+==========+=========+==================+
| 16#00FF_FFFF_0000_0000 | 8        | 7       | TRUE             |
+------------------------+----------+---------+------------------+
| 16#00FF_FFFF_0000_0000 | 8        | 6       | FALSE            |
+------------------------+----------+---------+------------------+
| 16#80FF_FFFF_0000_0000 | 8        | 7       | FALSE            |
+------------------------+----------+---------+------------------+
| 16#0000_0000_0000_FFFF | 8        | 2       | TRUE             |
+------------------------+----------+---------+------------------+
| 16#0000_0000_0000_FFFF | 8        | 1       | FALSE            |
+------------------------+----------+---------+------------------+
| 16#70FF_FFFF_FFFF_FFFF | 8        | 8       | TRUE             |
+------------------------+----------+---------+------------------+

.. <legal notes>

legal notes
=================
| SPDX-FileCopyrightText: © 2022 ekvip automation GmbH <info@ekvip.de>
| SPDX-License-Identifier: Apache-2.0
| For details check: Apache-2.0_

.. _Apache-2.0: https://www.apache.org/licenses/LICENSE-2.0

.. </legal notes>

parameters
=================
:return: ``TRUE`` all bytes are zero, ``FALSE`` at least one byte isn't zero

*)

METHOD PROTECTED isDataZero :BOOL
VAR_INPUT
	(* current binary data *)
	data			:POINTER TO BYTE;
	(* size to compare in bytes *)
	size			:DINT;
	(* last address to comapre *)
	end				:LINT;	
END_VAR
VAR
	isPointerAligned			:BOOL;
	remainingBytes				:DINT;
END_VAR
isPointerAligned := THIS^.isPointerAligend(data);

IF (isPointerAligned AND ((size-end) >= THIS^.REGISTER_SIZE)) THEN;
	remainingBytes := THIS^.getRemainingBytes(size);
	IF (remainingBytes > THIS^.ZERO_SIZE) THEN
		isDataZero := THIS^.isDataZeroBytewise(
			data := data,
			size := size,
			end := (size - remainingBytes)
		);
		RETURN (NOT isDataZero);
	END_IF
	isDataZero := THIS^.isDataZeroRegisterwise(
		data := data,
		size := (size - remainingBytes),
		end := end
	);	
ELSE	
	isDataZero := THIS^.isDataZeroBytewise(
		data := data,
		size := size,
		end := end
	);
END_IF;
END_METHOD

(*

short summary
=================
This method checks if the data of a byte pointer is zero through all bytes form (``size-1``) to ``end``.
The table below shows how it works.

+------------------------+----------+---------+------------------+
|    **value of data**   | **size** | **end** | **return value** |
+========================+==========+=========+==================+
| 16#00FF_FFFF_0000_0000 | 8        | 7       | TRUE             |
+------------------------+----------+---------+------------------+
| 16#00FF_FFFF_0000_0000 | 8        | 6       | FALSE            |
+------------------------+----------+---------+------------------+
| 16#80FF_FFFF_0000_0000 | 8        | 7       | FALSE            |
+------------------------+----------+---------+------------------+
| 16#0000_0000_0000_FFFF | 8        | 2       | TRUE             |
+------------------------+----------+---------+------------------+
| 16#0000_0000_0000_FFFF | 8        | 1       | FALSE            |
+------------------------+----------+---------+------------------+
| 16#70FF_FFFF_FFFF_FFFF | 8        | 8       | TRUE             |
+------------------------+----------+---------+------------------+

.. <legal notes>

legal notes
=================
| SPDX-FileCopyrightText: © 2022 ekvip automation GmbH <info@ekvip.de>
| SPDX-License-Identifier: Apache-2.0
| For details check: Apache-2.0_

.. _Apache-2.0: https://www.apache.org/licenses/LICENSE-2.0

.. </legal notes>

parameters
=================
:return: ``TRUE`` all bytes are zero, ``FALSE`` at least one byte isn't zero

*)

METHOD PROTECTED isDataZeroBytewise :BOOL
VAR_INPUT
	(* current binary data *)
	data			:POINTER TO BYTE;
	(* size to compare in bytes *)
	size			:DINT;
	(* last index to comapre *)
	end				:LINT;
END_VAR
VAR
	(* index of the current address *)
	pointerIndex	:LINT;
END_VAR
VAR CONSTANT
	NULL			:BYTE := 16#00;
END_VAR
isDataZeroBytewise := TRUE;

FOR pointerIndex := (size-1) TO end BY THIS^.DIRECTION_LE DO
	IF (data[pointerIndex] <> NULL) THEN
		isDataZeroBytewise := FALSE;
		RETURN;
	END_IF
END_FOR;
END_METHOD

(*

short summary
=================
This method checks if the data of a ``__XWORD pointer`` is zero
through all bytes form (``size-1``) to ``end``.

.. <legal notes>

legal notes
=================
| SPDX-FileCopyrightText: © 2022 ekvip automation GmbH <info@ekvip.de>
| SPDX-License-Identifier: Apache-2.0
| For details check: Apache-2.0_

.. _Apache-2.0: https://www.apache.org/licenses/LICENSE-2.0

.. </legal notes>

parameters
=================
:return: ``TRUE`` all bytes are zero, ``FALSE`` at least one byte isn't zero

*)

METHOD PROTECTED isDataZeroRegisterwise :BOOL
VAR_INPUT
	(* current binary data *)
	data			:POINTER TO __XWORD;
	(* size to compare in bytes *)
	size			:DINT;
	(* last address to comapre *)
	end				:LINT;
END_VAR
VAR
	(* index of the current address *)
	pointerIndex	:LINT;
END_VAR
VAR CONSTANT
	NULL			:__XWORD := 0;
END_VAR
isDataZeroRegisterwise := TRUE;

FOR pointerIndex := (size-1) TO end BY THIS^.DIRECTION_LE DO
	IF (data[pointerIndex] <> NULL) THEN
		isDataZeroRegisterwise := FALSE;
		RETURN;
	END_IF
END_FOR;
END_METHOD

(*

short summary
=================
This assertion method checks if all bytes of memory of
``data`` and ``dataToCompare`` are equal

.. attention:: 
	Binary comparison means it compares values byte by byte, regardless of type information (signs, ``REAL`` etc...)
	and it compares padding bytes, too.

.. attention:: 
	``STRING`` and ``WSTRING`` is null terminated
	that means TwinCAT sets null byte/word at the end of the string and touches nothing else
	For example ``foo :STRING(3) := 'foo';`` looks binary 16#66 16#6F 16#6F 16#00.
	if you set foo to an empty string ``foo := ''`` it looks like 16#00 16#6F 16#6F 16#00.

.. attention:: 
	It works not for bits because the minimum size must be at least one byte. If the ``__SYSTEM.TYPE_CLASS``
	of ``data`` ``AND`` ``dataToCompare is ``__SYSTEM.TYPE_CLASS.TYPE_BOOL`` ``OR`` ``__SYSTEM.TYPE_CLASS.TYPE_BIT``
	it uses the ``TO_BOOL`` operator for comarison. That means for ``__SYSTEM.TYPE_CLASS.TYPE_BIT`` it has no idea
	if the single ``BIT`` is set or unset, it compares just the whole ``BYTE``.

.. <legal notes>

legal notes
=================
| SPDX-FileCopyrightText: © 2022 ekvip automation GmbH <info@ekvip.de>
| SPDX-License-Identifier: Apache-2.0
| For details check: Apache-2.0_

.. _Apache-2.0: https://www.apache.org/licenses/LICENSE-2.0

.. </legal notes>

parameters
=================

*)

METHOD isEqualTo
VAR_INPUT
	(* current binary data *)
	data			:ANY;
	(* binary data with the expected values *)
	dataToCompare	:ANY;
	(* message if the assertion is false *)
	message			:AssertMessage;
END_VAR
IF (THIS^.binaryCompare(data, dataToCompare) <> CNM_ReturnTypes.ComparationResult.EQUAL) THEN
	THIS^.assertionWasWrong(message, THIS^.getDebugInfo('isEqualTo'));
END_IF
END_METHOD

(*

short summary
=================
This assertion method checks the bytes of memory of
``data`` and ``dataToCompare`` if the content of the first unequal
``data`` byte is greater than the byte of ``dataToCompare``
the assertion is true. Direction of comaprison is little endian.

.. attention:: 
	Binary comparison means it compares values byte by byte, regardless of type information (signs, ``REAL`` etc...)
	and it compares padding bytes, too.

.. attention:: 
	``STRING`` and ``WSTRING`` is null terminated
	that means TwinCAT sets null byte/word at the end of the string and touches nothing else
	For example ``foo :STRING(3) := 'foo';`` looks binary 16#66 16#6F 16#6F 16#00.
	if you set foo to an empty string ``foo := ''`` it looks like 16#00 16#6F 16#6F 16#00.

.. attention:: 
	It works not for bits because the minimum size must be at least one byte. If the ``__SYSTEM.TYPE_CLASS``
	of ``data`` ``AND`` ``dataToCompare is ``__SYSTEM.TYPE_CLASS.TYPE_BOOL`` ``OR`` ``__SYSTEM.TYPE_CLASS.TYPE_BIT``
	it uses the ``TO_BOOL`` operator for comarison. That means for ``__SYSTEM.TYPE_CLASS.TYPE_BIT`` it has no idea
	if the single ``BIT`` is set or unset, it compares just the whole ``BYTE``.

.. <legal notes>

legal notes
=================
| SPDX-FileCopyrightText: © 2022 ekvip automation GmbH <info@ekvip.de>
| SPDX-License-Identifier: Apache-2.0
| For details check: Apache-2.0_

.. _Apache-2.0: https://www.apache.org/licenses/LICENSE-2.0

.. </legal notes>

parameters
=================

*)

METHOD isGreaterThan
VAR_INPUT
	(* current binary data *)
	data			:ANY;
	(* binary data with smaller values *)
	dataToCompare	:ANY;
	(* message if the assertion is false *)
	message			:AssertMessage;
END_VAR
IF (THIS^.binaryCompare(data, dataToCompare) <> CNM_ReturnTypes.ComparationResult.GREATER) THEN
	THIS^.assertionWasWrong(message, THIS^.getDebugInfo('isGreaterThan'));
END_IF
END_METHOD

(*

short summary
=================
This assertion method checks the bytes of memory of
``data`` and ``dataToCompare`` if the content of the first unequal
``data`` byte is less than the byte of ``dataToCompare``
the assertion is true. Direction of comaprison is little endian.

.. <legal notes>

.. attention:: 
	Binary comparison means it compares values byte by byte, regardless of type information (signs, ``REAL`` etc...)
	and it compares padding bytes, too.

.. attention:: 
	``STRING`` and ``WSTRING`` is null terminated
	that means TwinCAT sets null byte/word at the end of the string and touches nothing else
	For example ``foo :STRING(3) := 'foo';`` looks binary 16#66 16#6F 16#6F 16#00.
	if you set foo to an empty string ``foo := ''`` it looks like 16#00 16#6F 16#6F 16#00.

.. attention:: 
	It works not for bits because the minimum size must be at least one byte. If the ``__SYSTEM.TYPE_CLASS``
	of ``data`` ``AND`` ``dataToCompare is ``__SYSTEM.TYPE_CLASS.TYPE_BOOL`` ``OR`` ``__SYSTEM.TYPE_CLASS.TYPE_BIT``
	it uses the ``TO_BOOL`` operator for comarison. That means for ``__SYSTEM.TYPE_CLASS.TYPE_BIT`` it has no idea
	if the single ``BIT`` is set or unset, it compares just the whole ``BYTE``.

legal notes
=================
| SPDX-FileCopyrightText: © 2022 ekvip automation GmbH <info@ekvip.de>
| SPDX-License-Identifier: Apache-2.0
| For details check: Apache-2.0_

.. _Apache-2.0: https://www.apache.org/licenses/LICENSE-2.0

.. </legal notes>

parameters
=================

*)

METHOD isLessThan
VAR_INPUT
	(* current binary data *)
	data			:ANY;
	(* binary data with greater values *)
	dataToCompare	:ANY;
	(* message if the assertion is false *)
	message			:AssertMessage;
END_VAR
IF (THIS^.binaryCompare(data, dataToCompare) <> CNM_ReturnTypes.ComparationResult.SMALLER) THEN
	THIS^.assertionWasWrong(message, THIS^.getDebugInfo('isLessThan'));
END_IF
END_METHOD

(*

short summary
=================
This assertion method checks if minimal one byte of memory of
``data`` and ``dataToCompare`` is not equal

.. attention:: 
	Binary comparison means it compares values byte by byte, regardless of type information (signs, ``REAL`` etc...)
	and it compares padding bytes, too.

.. attention:: 
	``STRING`` and ``WSTRING`` is null terminated
	that means TwinCAT sets null byte/word at the end of the string and touches nothing else
	For example ``foo :STRING(3) := 'foo';`` looks binary 16#66 16#6F 16#6F 16#00.
	if you set foo to an empty string ``foo := ''`` it looks like 16#00 16#6F 16#6F 16#00.

.. attention:: 
	It works not for bits because the minimum size must be at least one byte. If the ``__SYSTEM.TYPE_CLASS``
	of ``data`` ``AND`` ``dataToCompare is ``__SYSTEM.TYPE_CLASS.TYPE_BOOL`` ``OR`` ``__SYSTEM.TYPE_CLASS.TYPE_BIT``
	it uses the ``TO_BOOL`` operator for comarison. That means for ``__SYSTEM.TYPE_CLASS.TYPE_BIT`` it has no idea
	if the single ``BIT`` is set or unset, it compares just the whole ``BYTE``.

.. <legal notes>

legal notes
=================
| SPDX-FileCopyrightText: © 2022 ekvip automation GmbH <info@ekvip.de>
| SPDX-License-Identifier: Apache-2.0
| For details check: Apache-2.0_

.. _Apache-2.0: https://www.apache.org/licenses/LICENSE-2.0

.. </legal notes>

parameters
=================

*)

METHOD isNotEqualTo
VAR_INPUT
	(* current binary data *)
	data			:ANY;
	(* binary data with the unexpected values *)
	dataToCompare	:ANY;
	(* message if the assertion is false *)
	message			:AssertMessage;
END_VAR
IF (THIS^.binaryCompare(data, dataToCompare) = CNM_ReturnTypes.ComparationResult.EQUAL) THEN
	THIS^.assertionWasWrong(message, THIS^.getDebugInfo('isNotEqualTo'));
END_IF
END_METHOD

(*

short summary
=================
This method checks if an address is aligned to a register

.. <legal notes>

legal notes
=================
| SPDX-FileCopyrightText: © 2022 ekvip automation GmbH <info@ekvip.de>
| SPDX-License-Identifier: Apache-2.0
| For details check: Apache-2.0_

.. _Apache-2.0: https://www.apache.org/licenses/LICENSE-2.0

.. </legal notes>

parameters
=================
:return: ``TRUE`` pointer address **is** aligned to a register,
``FALSE`` pointer address **isn't** aligned to a register

*)

METHOD PROTECTED isPointerAligend :BOOL
VAR_INPUT
	(* address to check *)
	in :PVOID;
END_VAR
VAR CONSTANT
	(* 
	for 32 bit systems address is aligned if 2#111 is unset,
	for 64 bit systems address is aligned if 2#1111 is unset
	*)
	ALIGNMENT_MASK	:__XWORD := (SIZEOF(__XWORD)-1);
	(* just to check if relevant bits unset *)
	WELL_ALIGNED	:__XWORD := 0;
END_VAR
isPointerAligend := ((in AND ALIGNMENT_MASK) = WELL_ALIGNED);
END_METHOD

END_FUNCTION_BLOCK

// ---- Assertor/classes/AbstactAssertion.TcPOU
(*

short summary
=================
This abstract class is for all the assertion classes to ease and unify
the callbacks

.. <legal notes>

legal notes
=================
| SPDX-FileCopyrightText: © 2022 ekvip automation GmbH <info@ekvip.de>
| SPDX-License-Identifier: Apache-2.0
| For details check: Apache-2.0_

.. _Apache-2.0: https://www.apache.org/licenses/LICENSE-2.0

.. </legal notes>

methods and properties
=======================

*)

{attribute 'reflection'}
FUNCTION_BLOCK INTERNAL ABSTRACT AbstactAssertion EXTENDS CNM_AbstractObject.Object IMPLEMENTS IAssertCallBackSetter
VAR
	(* the class that must be informed if an assertion is false *)
	callBack	:IAssertCallback;
END_VAR

(*

short summary
=================
This method is called if an assertion was ``FALSE``

.. <legal notes>

legal notes
=================
| SPDX-FileCopyrightText: © 2022 ekvip automation GmbH <info@ekvip.de>
| SPDX-License-Identifier: Apache-2.0
| For details check: Apache-2.0_

.. _Apache-2.0: https://www.apache.org/licenses/LICENSE-2.0

.. </legal notes>

parameters
=================

*)

METHOD PROTECTED assertionWasWrong
VAR_INPUT
	(* alarm message *)
	message			:AssertMessage;
	(* debugging information *) 
	additionalText	:Tc2_System.T_MaxString;
END_VAR
IF (THIS^.isObjectValid(THIS^.callBack)) THEN
	THIS^.callBack.assertionWasWrong(
		caller			:= THIS^,
		message			:= message,
		additionalText	:= additionalText
	);
END_IF
END_METHOD

(*

short summary
=================
This abstract property returns the class name of the concrete object, 
It's for debugging purpose

.. attention:: 
	For derivations: **It is necessary that this property is overridden by the concrete class**

.. <legal notes>

legal notes
=================
| SPDX-FileCopyrightText: © 2022 ekvip automation GmbH <info@ekvip.de>
| SPDX-License-Identifier: Apache-2.0
| For details check: Apache-2.0_

.. _Apache-2.0: https://www.apache.org/licenses/LICENSE-2.0

.. </legal notes>

*)

PROPERTY ABSTRACT className : CNM_AbstractObject.ClassName
GET
END_GET
END_PROPERTY

(*

short summary
=================
This method returns a debug info string

.. <legal notes>

legal notes
=================
| SPDX-FileCopyrightText: © 2022 ekvip automation GmbH <info@ekvip.de>
| SPDX-License-Identifier: Apache-2.0
| For details check: Apache-2.0_

.. _Apache-2.0: https://www.apache.org/licenses/LICENSE-2.0

.. </legal notes>

parameters
=================
:return: debug info string, it contains the caller method name and the class name. 
Format is ``'ClassName.methodName: Assertion was false'``

*)

METHOD PROTECTED getDebugInfo :Tc2_System.T_MaxString
VAR_INPUT
	(* name of the caller method *) 
	caller	:Tc2_System.T_MaxString;
END_VAR
getDebugInfo := Tc2_Standard.CONCAT(
	THIS^.className,
	Tc2_Standard.CONCAT(
		'.',
		Tc2_Standard.CONCAT(
			caller,
			': Assertion was false'
		)
	)
);
END_METHOD

(*

short summary
=================
This methods is the setter for the callback class if an assertion was false

.. <legal notes>

legal notes
=================
| SPDX-FileCopyrightText: © 2022 ekvip automation GmbH <info@ekvip.de>
| SPDX-License-Identifier: Apache-2.0
| For details check: Apache-2.0_

.. _Apache-2.0: https://www.apache.org/licenses/LICENSE-2.0

.. </legal notes>

parameters
=================

*)

METHOD setCallBack
VAR_INPUT
	(* the class that must be informed if an assertion is false *)
	callBack	:IAssertCallback;  
END_VAR
THIS^.callBack := callBack;
END_METHOD

END_FUNCTION_BLOCK

// ---- Assertor/Assertions/BinaryAssertions/udfhgdshfksfkjshdkjfdhsfsdfsdfsfsdfsdfsdsdf.TcPOU
FUNCTION udfhgdshfksfkjshdkjfdhsfsdfsdfsfsdfsdfsdsdf : sdfdsfsdfsd
VAR_INPUT
END_VAR
VAR
END_VAR

END_FUNCTION

// ---- Assertor/Assertions/BitNumberAssertions/Byte/classes/ByteAssertions.TcPOU
(*

short summary
=================
This class provides assert statements for bytes.
It implements :ref:`IByteAssertions`

.. <legal notes>

legal notes
=================
| SPDX-FileCopyrightText: © 2022 ekvip automation GmbH <info@ekvip.de>
| SPDX-License-Identifier: Apache-2.0
| For details check: Apache-2.0_

.. _Apache-2.0: https://www.apache.org/licenses/LICENSE-2.0

.. </legal notes>

methods and properties
=======================

*)

{attribute 'reflection'}
FUNCTION_BLOCK INTERNAL ByteAssertions EXTENDS AbstactAssertion IMPLEMENTS IByteAssertions
VAR
END_VAR
VAR CONSTANT
	(* least significant bit *)
	LSB	:BYTE := 16#01;
	(* most significant bit *)
	MSB :BYTE := 16#80;
END_VAR

(*

short summary
=================
This assertion method checks if the result current value bitwise ``AND`` mask is equal to the expected value

.. <legal notes>

legal notes
=================
| SPDX-FileCopyrightText: © 2022 ekvip automation GmbH <info@ekvip.de>
| SPDX-License-Identifier: Apache-2.0
| For details check: Apache-2.0_

.. _Apache-2.0: https://www.apache.org/licenses/LICENSE-2.0

.. </legal notes>

parameters
=================

*)

METHOD andMaskIsEqualTo
VAR_INPUT
	(* current value to check *)
	currentValue	:BYTE;
	(* 2nd operand for bitwise operation *)
	mask			:BYTE;
	(* expected result after masking *)
	expectedValue	:BYTE;
	(* message if the assertion is false *)
	message			:AssertMessage;
END_VAR
IF ((currentValue AND mask) <> expectedValue) THEN
	THIS^.assertionWasWrong(message, THIS^.getDebugInfo('andMaskIsEqualTo'));
END_IF
END_METHOD

(*

short summary
=================
This assertion method checks if the result current value bitwise ``AND`` mask
is not equal to the unexpected value

.. <legal notes>

legal notes
=================
| SPDX-FileCopyrightText: © 2022 ekvip automation GmbH <info@ekvip.de>
| SPDX-License-Identifier: Apache-2.0
| For details check: Apache-2.0_

.. _Apache-2.0: https://www.apache.org/licenses/LICENSE-2.0

.. </legal notes>

parameters
=================

*)

METHOD andMaskIsNotEqualTo
VAR_INPUT
	(* current value to check *)
	currentValue	:BYTE;
	(* 2nd operand for bitwise operation *)
	mask			:BYTE;
	(* unexpected result after masking *)
	unexpectedValue	:BYTE;
	(* message if the assertion is false *)
	message			:AssertMessage;
END_VAR
IF ((currentValue AND mask) = unexpectedValue) THEN
	THIS^.assertionWasWrong(message, THIS^.getDebugInfo('andMaskIsNotEqualTo'));
END_IF
END_METHOD

(*

short summary
=================
This assertion method checks if the selected bit of current value
is equal to the expected value

.. <legal notes>

legal notes
=================
| SPDX-FileCopyrightText: © 2022 ekvip automation GmbH <info@ekvip.de>
| SPDX-License-Identifier: Apache-2.0
| For details check: Apache-2.0_

.. _Apache-2.0: https://www.apache.org/licenses/LICENSE-2.0

.. </legal notes>

parameters
=================

*)

METHOD bitXIsEqualTo
VAR_INPUT
	(* current value to check *)
	currentValue	:BYTE;
	(* number of bit to check *)
	number			:BitNumberByte;
	(* expected value of bit *)
	expectedValue	:BOOL;
	(* message if the assertion is false *)
	message			:AssertMessage;
END_VAR
IF (
	TO_BOOL(
		TO_BYTE(SHL(THIS^.LSB, number))
		AND currentValue
	) <> expectedValue
) THEN
	THIS^.assertionWasWrong(message, THIS^.getDebugInfo('bitXIsEqualTo'));
END_IF
END_METHOD

(*

short summary
=================
This assertion method checks if the selected bit of current value
is not equal to the unexpected value

.. <legal notes>

legal notes
=================
| SPDX-FileCopyrightText: © 2022 ekvip automation GmbH <info@ekvip.de>
| SPDX-License-Identifier: Apache-2.0
| For details check: Apache-2.0_

.. _Apache-2.0: https://www.apache.org/licenses/LICENSE-2.0

.. </legal notes>

parameters
=================

*)

METHOD bitXIsNotEqualTo
VAR_INPUT
	(* current value to check *)
	currentValue	:BYTE;
	(* number of bit to check *)
	number			:BitNumberByte;
	(* unexpected value of bit *)
	unexpectedValue	:BOOL;
	(* message if the assertion is false *)
	message			:AssertMessage;
END_VAR
IF (
	TO_BOOL(
		TO_BYTE(SHL(THIS^.LSB, number))
		AND currentValue
	) = unexpectedValue
) THEN
	THIS^.assertionWasWrong(message, THIS^.getDebugInfo('bitXIsNotEqualTo'));
END_IF
END_METHOD

(*

short summary
=================
This assertion method checks if the selected bit of current value
is set

.. <legal notes>

legal notes
=================
| SPDX-FileCopyrightText: © 2022 ekvip automation GmbH <info@ekvip.de>
| SPDX-License-Identifier: Apache-2.0
| For details check: Apache-2.0_

.. _Apache-2.0: https://www.apache.org/licenses/LICENSE-2.0

.. </legal notes>

parameters
=================

*)

METHOD bitXIsSet
VAR_INPUT
	(* current value to check *)
	currentValue	:BYTE;
	(* number of bit to check *)
	number			:BitNumberByte;
	(* message if the assertion is false *)
	message			:AssertMessage;
END_VAR
IF (
	NOT TO_BOOL(
		TO_BYTE(SHL(THIS^.LSB, number))
		AND currentValue
	)
) THEN
	THIS^.assertionWasWrong(message, THIS^.getDebugInfo('bitXIsSet'));
END_IF
END_METHOD

(*

short summary
=================
This assertion method checks if the selected bit of current value
is unset

.. <legal notes>

legal notes
=================
| SPDX-FileCopyrightText: © 2022 ekvip automation GmbH <info@ekvip.de>
| SPDX-License-Identifier: Apache-2.0
| For details check: Apache-2.0_

.. _Apache-2.0: https://www.apache.org/licenses/LICENSE-2.0

.. </legal notes>

parameters
=================

*)

METHOD bitXIsUnset
VAR_INPUT
	(* current value to check *)
	currentValue	:BYTE;
	(* number of bit to check *)
	number			:BitNumberByte;
	(* message if the assertion is false *)
	message			:AssertMessage;
END_VAR
IF (
	TO_BOOL(
		TO_BYTE(SHL(THIS^.LSB, number))
		AND currentValue
	)
) THEN
	THIS^.assertionWasWrong(message, THIS^.getDebugInfo('bitXIsUnset'));
END_IF
END_METHOD

(*

short summary
=================
This abstract property returns the class name of the concrete object, 
It's for debugging purpose

.. <legal notes>

legal notes
=================
| SPDX-FileCopyrightText: © 2022 ekvip automation GmbH <info@ekvip.de>
| SPDX-License-Identifier: Apache-2.0
| For details check: Apache-2.0_

.. _Apache-2.0: https://www.apache.org/licenses/LICENSE-2.0

.. </legal notes>

*)

PROPERTY className :CNM_AbstractObject.ClassName
GET
className := 'CNM_AssertionInterfaceLib.ByteAssertions';
END_GET
END_PROPERTY

(*

short summary
=================
This assertion method checks if the least significant bit of current value
is equal to the expected value

.. <legal notes>

legal notes
=================
| SPDX-FileCopyrightText: © 2022 ekvip automation GmbH <info@ekvip.de>
| SPDX-License-Identifier: Apache-2.0
| For details check: Apache-2.0_

.. _Apache-2.0: https://www.apache.org/licenses/LICENSE-2.0

.. </legal notes>

parameters
=================

*)

METHOD lsbIsEqualTo
VAR_INPUT
	(* current value to check *)
	currentValue	:BYTE;
	(* expected value of lsb *)
	expectedValue	:BOOL;
	(* message if the assertion is false *)
	message			:AssertMessage;
END_VAR
IF (TO_BOOL(currentValue AND THIS^.LSB) <> expectedValue) THEN
	THIS^.assertionWasWrong(message, THIS^.getDebugInfo('lsbIsEqualTo'));
END_IF
END_METHOD

(*

short summary
=================
This assertion method checks if the least significant bit of current value
is not equal to the unexpected value

.. <legal notes>

legal notes
=================
| SPDX-FileCopyrightText: © 2022 ekvip automation GmbH <info@ekvip.de>
| SPDX-License-Identifier: Apache-2.0
| For details check: Apache-2.0_

.. _Apache-2.0: https://www.apache.org/licenses/LICENSE-2.0

.. </legal notes>

parameters
=================

*)

METHOD lsbIsNotEqualTo
VAR_INPUT
	(* current value to check *)
	currentValue	:BYTE;
	(* unexpected value of lsb *)
	unexpectedValue	:BOOL;
	(* message if the assertion is false *)
	message			:AssertMessage;
END_VAR
IF (TO_BOOL(currentValue AND THIS^.LSB) = unexpectedValue) THEN
	THIS^.assertionWasWrong(message, THIS^.getDebugInfo('lsbIsNotEqualTo'));
END_IF
END_METHOD

(*

short summary
=================
This assertion method checks if the least significant bit of current value
is set

.. <legal notes>

legal notes
=================
| SPDX-FileCopyrightText: © 2022 ekvip automation GmbH <info@ekvip.de>
| SPDX-License-Identifier: Apache-2.0
| For details check: Apache-2.0_

.. _Apache-2.0: https://www.apache.org/licenses/LICENSE-2.0

.. </legal notes>

parameters
=================

*)

METHOD lsbIsSet
VAR_INPUT
	(* current value to check *)
	currentValue	:BYTE;
	(* message if the assertion is false *)
	message			:AssertMessage;
END_VAR
IF (NOT TO_BOOL(currentValue AND THIS^.LSB)) THEN
	THIS^.assertionWasWrong(message, THIS^.getDebugInfo('lsbIsSet'));
END_IF
END_METHOD

(*

short summary
=================
This assertion method checks if the least significant bit of current value
is unset

.. <legal notes>

legal notes
=================
| SPDX-FileCopyrightText: © 2022 ekvip automation GmbH <info@ekvip.de>
| SPDX-License-Identifier: Apache-2.0
| For details check: Apache-2.0_

.. _Apache-2.0: https://www.apache.org/licenses/LICENSE-2.0

.. </legal notes>

parameters
=================

*)

METHOD lsbIsUnset
VAR_INPUT
	(* current value to check *)
	currentValue	:BYTE;
	(* message if the assertion is false *)
	message			:AssertMessage;
END_VAR
IF (TO_BOOL(currentValue AND THIS^.LSB)) THEN
	THIS^.assertionWasWrong(message, THIS^.getDebugInfo('lsbIsUnset'));
END_IF
END_METHOD

(*

short summary
=================
This assertion method checks if the most significant bit of current value
is equal to the expected value

.. <legal notes>

legal notes
=================
| SPDX-FileCopyrightText: © 2022 ekvip automation GmbH <info@ekvip.de>
| SPDX-License-Identifier: Apache-2.0
| For details check: Apache-2.0_

.. _Apache-2.0: https://www.apache.org/licenses/LICENSE-2.0

.. </legal notes>

parameters
=================

*)

METHOD msbIsEqualTo
VAR_INPUT
	(* current value to check *)
	currentValue	:BYTE;
	(* expected value of msb *)
	expectedValue	:BOOL;
	(* message if the assertion is false *)
	message			:AssertMessage;
END_VAR
IF (TO_BOOL(currentValue AND THIS^.MSB) <> expectedValue) THEN
	THIS^.assertionWasWrong(message, THIS^.getDebugInfo('msbIsEqualTo'));
END_IF
END_METHOD

(*

short summary
=================
This assertion method checks if the most significant bit of current value
is not equal to the unexpected value

.. <legal notes>

legal notes
=================
| SPDX-FileCopyrightText: © 2022 ekvip automation GmbH <info@ekvip.de>
| SPDX-License-Identifier: Apache-2.0
| For details check: Apache-2.0_

.. _Apache-2.0: https://www.apache.org/licenses/LICENSE-2.0

.. </legal notes>

parameters
=================

*)

METHOD msbIsNotEqualTo
VAR_INPUT
	(* current value to check *)
	currentValue	:BYTE;
	(* unexpected value of msb *)
	unexpectedValue	:BOOL;
	(* message if the assertion is false *)
	message			:AssertMessage;
END_VAR
IF (TO_BOOL(currentValue AND THIS^.MSB) = unexpectedValue) THEN
	THIS^.assertionWasWrong(message, THIS^.getDebugInfo('msbIsNotEqualTo'));
END_IF
END_METHOD

(*

short summary
=================
This assertion method checks if the most significant bit of current value
is set

.. <legal notes>

legal notes
=================
| SPDX-FileCopyrightText: © 2022 ekvip automation GmbH <info@ekvip.de>
| SPDX-License-Identifier: Apache-2.0
| For details check: Apache-2.0_

.. _Apache-2.0: https://www.apache.org/licenses/LICENSE-2.0

.. </legal notes>

parameters
=================

*)

METHOD msbIsSet
VAR_INPUT
	(* current value to check *)
	currentValue	:BYTE;
	(* message if the assertion is false *)
	message			:AssertMessage;
END_VAR
IF (NOT TO_BOOL(currentValue AND THIS^.MSB)) THEN
	THIS^.assertionWasWrong(message, THIS^.getDebugInfo('msbIsSet'));
END_IF
END_METHOD

(*

short summary
=================
This assertion method checks if the most significant bit of current value
is unset

.. <legal notes>

legal notes
=================
| SPDX-FileCopyrightText: © 2022 ekvip automation GmbH <info@ekvip.de>
| SPDX-License-Identifier: Apache-2.0
| For details check: Apache-2.0_

.. _Apache-2.0: https://www.apache.org/licenses/LICENSE-2.0

.. </legal notes>

parameters
=================

*)

METHOD msbIsUnset
VAR_INPUT
	(* current value to check *)
	currentValue	:BYTE;
	(* message if the assertion is false *)
	message			:AssertMessage;
END_VAR
IF (TO_BOOL(currentValue AND THIS^.MSB)) THEN
	THIS^.assertionWasWrong(message, THIS^.getDebugInfo('msbIsUnset'));
END_IF
END_METHOD

(*

short summary
=================
This assertion method checks if the result current value bitwise ``OR`` mask is equal to the expected value

.. <legal notes>

legal notes
=================
| SPDX-FileCopyrightText: © 2022 ekvip automation GmbH <info@ekvip.de>
| SPDX-License-Identifier: Apache-2.0
| For details check: Apache-2.0_

.. _Apache-2.0: https://www.apache.org/licenses/LICENSE-2.0

.. </legal notes>

parameters
=================

*)

METHOD orMaskIsEqualTo
VAR_INPUT
	(* current value to check *)
	currentValue	:BYTE;
	(* 2nd operand for bitwise operation *)
	mask			:BYTE;
	(* expected result after masking *)
	expectedValue	:BYTE;
	(* message if the assertion is false *)
	message			:AssertMessage;
END_VAR
IF ((currentValue OR mask) <> expectedValue) THEN
	THIS^.assertionWasWrong(message, THIS^.getDebugInfo('orMaskIsEqualTo'));
END_IF
END_METHOD

(*

short summary
=================
This assertion method checks if the result current value bitwise ``OR`` mask 
is not equal to the unexpected value

.. <legal notes>

legal notes
=================
| SPDX-FileCopyrightText: © 2022 ekvip automation GmbH <info@ekvip.de>
| SPDX-License-Identifier: Apache-2.0
| For details check: Apache-2.0_

.. _Apache-2.0: https://www.apache.org/licenses/LICENSE-2.0

.. </legal notes>

parameters
=================

*)

METHOD orMaskIsNotEqualTo
VAR_INPUT
	(* current value to check *)
	currentValue	:BYTE;
	(* 2nd operand for bitwise operation *)
	mask			:BYTE;
	(* unexpected result after masking *)
	unexpectedValue	:BYTE;
	(* message if the assertion is false *)
	message			:AssertMessage;
END_VAR
IF ((currentValue OR mask) = unexpectedValue) THEN
	THIS^.assertionWasWrong(message, THIS^.getDebugInfo('orMaskIsNotEqualTo'));
END_IF
END_METHOD

(*

short summary
=================
This assertion method checks if the current value is equal to the expected value

.. <legal notes>

legal notes
=================
| SPDX-FileCopyrightText: © 2022 ekvip automation GmbH <info@ekvip.de>
| SPDX-License-Identifier: Apache-2.0
| For details check: Apache-2.0_

.. _Apache-2.0: https://www.apache.org/licenses/LICENSE-2.0

.. </legal notes>

parameters
=================

*)

METHOD valueIsEqualTo
VAR_INPUT
	(* current value to check *)
	currentValue	:BYTE;
	(* expected value to compare *)
	expectedValue	:BYTE;
	(* message if the assertion is false *)
	message			:AssertMessage;
END_VAR
IF (currentValue <> expectedValue) THEN
	THIS^.assertionWasWrong(message, THIS^.getDebugInfo('valueIsEqualTo'));
END_IF
END_METHOD

(*

short summary
=================
This assertion method checks if the current value is greater than the less value

.. <legal notes>

legal notes
=================
| SPDX-FileCopyrightText: © 2022 ekvip automation GmbH <info@ekvip.de>
| SPDX-License-Identifier: Apache-2.0
| For details check: Apache-2.0_

.. _Apache-2.0: https://www.apache.org/licenses/LICENSE-2.0

.. </legal notes>

parameters
=================

*)

METHOD valueIsGreaterThan
VAR_INPUT
	(* current value to check *)
	currentValue	:BYTE;
	(* less than lower limit *)
	lessValue		:BYTE;
	(* message if the assertion is false *)
	message			:AssertMessage;
END_VAR
IF (currentValue <= lessValue) THEN
	THIS^.assertionWasWrong(message, THIS^.getDebugInfo('valueIsGreaterThan'));
END_IF
END_METHOD

(*

short summary
=================
This assertion method checks if the current value is inside a limit

.. attention:: 
	limits are included: ``valueIsInRangeOf(3, 3, 3)`` is a true assertion

.. <legal notes>

legal notes
=================
| SPDX-FileCopyrightText: © 2022 ekvip automation GmbH <info@ekvip.de>
| SPDX-License-Identifier: Apache-2.0
| For details check: Apache-2.0_

.. _Apache-2.0: https://www.apache.org/licenses/LICENSE-2.0

.. </legal notes>

parameters
=================

*)

METHOD valueIsInRangeOf
VAR_INPUT
	(* lower limit for the current value *)
	lowerLimit		:BYTE;
	(* current value to check *)
	currentValue	:BYTE;
	(* upper limit for the current value *)
	upperLimit		:BYTE;
	(* message if the assertion is false *)
	message			:AssertMessage;
END_VAR
IF (
	(currentValue < lowerLimit)
	OR (currentValue > upperLimit)
) THEN
	THIS^.assertionWasWrong(message, THIS^.getDebugInfo('valueIsInRangeOf'));
END_IF
END_METHOD

(*

short summary
=================
This assertion method checks if the current value is less than the greater value

.. <legal notes>

legal notes
=================
| SPDX-FileCopyrightText: © 2022 ekvip automation GmbH <info@ekvip.de>
| SPDX-License-Identifier: Apache-2.0
| For details check: Apache-2.0_

.. _Apache-2.0: https://www.apache.org/licenses/LICENSE-2.0

.. </legal notes>

parameters
=================

*)

METHOD valueIsLessThan
VAR_INPUT
	(* current value to check *)
	currentValue	:BYTE;
	(* greater than upper limit *)
	greaterValue	:BYTE;
	(* message if the assertion is false *)
	message			:AssertMessage;
END_VAR
IF (currentValue >= greaterValue) THEN
	THIS^.assertionWasWrong(message, THIS^.getDebugInfo('valueIsLessThan'));
END_IF
END_METHOD

(*

short summary
=================
This assertion method checks if the current value is less than or equal to the maximum value

.. <legal notes>

legal notes
=================
| SPDX-FileCopyrightText: © 2022 ekvip automation GmbH <info@ekvip.de>
| SPDX-License-Identifier: Apache-2.0
| For details check: Apache-2.0_

.. _Apache-2.0: https://www.apache.org/licenses/LICENSE-2.0

.. </legal notes>

parameters
=================

*)

METHOD valueIsMax
VAR_INPUT
	(* current value to check *)
	currentValue	:BYTE;
	(* upper limit for the current value *)
	maximumValue	:BYTE;
	(* message if the assertion is false *)
	message			:AssertMessage;
END_VAR
IF (currentValue > maximumValue) THEN
	THIS^.assertionWasWrong(message, THIS^.getDebugInfo('valueIsMax'));
END_IF
END_METHOD

(*

short summary
=================
This assertion method checks if the current value is greater than or equal to the minimum value

.. <legal notes>

legal notes
=================
| SPDX-FileCopyrightText: © 2022 ekvip automation GmbH <info@ekvip.de>
| SPDX-License-Identifier: Apache-2.0
| For details check: Apache-2.0_

.. _Apache-2.0: https://www.apache.org/licenses/LICENSE-2.0

.. </legal notes>

parameters
=================

*)

METHOD valueIsMin
VAR_INPUT
	(* current value to check *)
	currentValue	:BYTE;
	(* lower limit for the current value *)
	minimumValue	:BYTE;
	(* message if the assertion is false *)
	message			:AssertMessage;
END_VAR
IF (currentValue < minimumValue) THEN
	THIS^.assertionWasWrong(message, THIS^.getDebugInfo('valueIsMin'));
END_IF
END_METHOD

(*

short summary
=================
This assertion method checks if the current value is not equal to the unexpected value

.. <legal notes>

legal notes
=================
| SPDX-FileCopyrightText: © 2022 ekvip automation GmbH <info@ekvip.de>
| SPDX-License-Identifier: Apache-2.0
| For details check: Apache-2.0_

.. _Apache-2.0: https://www.apache.org/licenses/LICENSE-2.0

.. </legal notes>

parameters
=================

*)

METHOD valueIsNotEqualTo
VAR_INPUT
	(* current value to check *)
	currentValue	:BYTE;
	(* unexpected value to compare *)
	unexpectedValue	:BYTE;
	(* message if the assertion is false *)
	message			:AssertMessage;
END_VAR
IF (currentValue = unexpectedValue) THEN
	THIS^.assertionWasWrong(message, THIS^.getDebugInfo('valueIsNotEqualTo'));
END_IF
END_METHOD

(*

short summary
=================
This assertion method checks if the result current value bitwise ``XOR`` mask is equal to the expected value

.. <legal notes>

legal notes
=================
| SPDX-FileCopyrightText: © 2022 ekvip automation GmbH <info@ekvip.de>
| SPDX-License-Identifier: Apache-2.0
| For details check: Apache-2.0_

.. _Apache-2.0: https://www.apache.org/licenses/LICENSE-2.0

.. </legal notes>

parameters
=================

*)

METHOD xorMaskIsEqualTo
VAR_INPUT
	(* current value to check *)
	currentValue	:BYTE;
	(* 2nd operand for bitwise operation *)
	mask			:BYTE;
	(* expected result after masking *)
	expectedValue	:BYTE;
	(* message if the assertion is false *)
	message			:AssertMessage;
END_VAR
IF ((currentValue XOR mask) <> expectedValue) THEN
	THIS^.assertionWasWrong(message, THIS^.getDebugInfo('xorMaskIsEqualTo'));
END_IF
END_METHOD

(*

short summary
=================
This assertion method checks if the result current value bitwise ``XOR`` mask 
is not equal to the unexpected value

.. <legal notes>

legal notes
=================
| SPDX-FileCopyrightText: © 2022 ekvip automation GmbH <info@ekvip.de>
| SPDX-License-Identifier: Apache-2.0
| For details check: Apache-2.0_

.. _Apache-2.0: https://www.apache.org/licenses/LICENSE-2.0

.. </legal notes>

parameters
=================

*)

METHOD xorMaskIsNotEqualTo
VAR_INPUT
	(* current value to check *)
	currentValue	:BYTE;
	(* 2nd operand for bitwise operation *)
	mask			:BYTE;
	(* unexpected result after masking *)
	unexpectedValue	:BYTE;
	(* message if the assertion is false *)
	message			:AssertMessage;
END_VAR
IF ((currentValue XOR mask) = unexpectedValue) THEN
	THIS^.assertionWasWrong(message, THIS^.getDebugInfo('xorMaskIsNotEqualTo'));
END_IF
END_METHOD

END_FUNCTION_BLOCK

// ---- Assertor/Assertions/BitNumberAssertions/classes/BitNumberAssertions.TcPOU
(*

short summary
=================
| This class provides assert statements for bit numbers:
| It implements the interface :ref:`IBitNumberAssertions`
| For ``BYTE`` use :ref:`BitNumberAssertions.short`
| For ``WORD`` use :ref:`BitNumberAssertions.simple`
| For ``DWORD`` use :ref:`BitNumberAssertions.double`
| For ``LWORD`` use :ref:`BitNumberAssertions.long`
| For ``__XWORD`` use :ref:`BitNumberAssertions.x`

.. <legal notes>

legal notes
=================
| SPDX-FileCopyrightText: © 2022 ekvip automation GmbH <info@ekvip.de>
| SPDX-License-Identifier: Apache-2.0
| For details check: Apache-2.0_

.. _Apache-2.0: https://www.apache.org/licenses/LICENSE-2.0

.. </legal notes>

methods and properties
=======================

*)

{attribute 'reflection'}
FUNCTION_BLOCK INTERNAL BitNumberAssertions 
EXTENDS CNM_AbstractObject.Object 
IMPLEMENTS IBitNumberAssertions, IAssertCallBacksetter
VAR
	(* class to handle byte assertions *)
	byteAssertions	:ByteAssertions();
	(* class to handle word assertions *)
	wordAssertions	:WordAssertions();
	(* class to handle dword assertions *)
	dwordAssertions	:DWordAssertions();
	(* class to handle lword assertions *)
	lwordAssertions	:LWordAssertions();
	(* class to handle xword assertions *)
	xwordAssertions	:XWordAssertions();
END_VAR

(*

short summary
=================
This abstract property returns the class name of the concrete object, 
It's for debugging purpose

.. <legal notes>

legal notes
=================
| SPDX-FileCopyrightText: © 2022 ekvip automation GmbH <info@ekvip.de>
| SPDX-License-Identifier: Apache-2.0
| For details check: Apache-2.0_

.. _Apache-2.0: https://www.apache.org/licenses/LICENSE-2.0

.. </legal notes>

*)

PROPERTY className :CNM_AbstractObject.ClassName
GET
className := 'CNM_AssertionInterfaceLib.BitNumberAssertions';
END_GET
END_PROPERTY

(*

short summary
=================
Returns the interface :ref:`IDwordAssertions`
with assert statements for double words ``DWORD`` 

.. <legal notes>

legal notes
=================
| SPDX-FileCopyrightText: © 2022 ekvip automation GmbH <info@ekvip.de>
| SPDX-License-Identifier: Apache-2.0
| For details check: Apache-2.0_

.. _Apache-2.0: https://www.apache.org/licenses/LICENSE-2.0

.. </legal notes>

*)

PROPERTY double :IDwordAssertions
GET
double := THIS^.dwordAssertions;
END_GET
END_PROPERTY

(*

short summary
=================
Returns the interface :ref:`ILwordAssertions`
with assert statements for long words ``LWORD`` 

.. <legal notes>

legal notes
=================
| SPDX-FileCopyrightText: © 2022 ekvip automation GmbH <info@ekvip.de>
| SPDX-License-Identifier: Apache-2.0
| For details check: Apache-2.0_

.. _Apache-2.0: https://www.apache.org/licenses/LICENSE-2.0

.. </legal notes>

*)

PROPERTY long :ILwordAssertions
GET
long := THIS^.lwordAssertions;
END_GET
END_PROPERTY

(*

short summary
=================
This methods is the setter for the callback class if an assertion was false

.. <legal notes>

legal notes
=================
| SPDX-FileCopyrightText: © 2022 ekvip automation GmbH <info@ekvip.de>
| SPDX-License-Identifier: Apache-2.0
| For details check: Apache-2.0_

.. _Apache-2.0: https://www.apache.org/licenses/LICENSE-2.0

.. </legal notes>

parameters
=================

*)

METHOD setCallBack
VAR_INPUT
	(* the class that must be informed if an assertion is false *)
	callBack	:IAssertCallback;  
END_VAR
THIS^.byteAssertions.setCallBack(callBack);
THIS^.wordAssertions.setCallBack(callBack);
THIS^.dwordAssertions.setCallBack(callBack);
THIS^.lwordAssertions.setCallBack(callBack);
THIS^.xwordAssertions.setCallBack(callBack);
END_METHOD

(*

short summary
=================
Returns the interface :ref:`IByteAssertions`
with assert statements for bytes

.. <legal notes>

legal notes
=================
| SPDX-FileCopyrightText: © 2022 ekvip automation GmbH <info@ekvip.de>
| SPDX-License-Identifier: Apache-2.0
| For details check: Apache-2.0_

.. _Apache-2.0: https://www.apache.org/licenses/LICENSE-2.0

.. </legal notes>

*)

PROPERTY short :IByteAssertions
GET
short := THIS^.byteAssertions;
END_GET
END_PROPERTY

(*

short summary
=================
Returns the interface :ref:`IWordAssertions`
with assert statements for words 

.. <legal notes>

legal notes
=================
| SPDX-FileCopyrightText: © 2022 ekvip automation GmbH <info@ekvip.de>
| SPDX-License-Identifier: Apache-2.0
| For details check: Apache-2.0_

.. _Apache-2.0: https://www.apache.org/licenses/LICENSE-2.0

.. </legal notes>

*)

PROPERTY simple :IWordAssertions
GET
simple := THIS^.wordAssertions;
END_GET
END_PROPERTY

(*

short summary
=================
Returns the interface :ref:`IXwordAssertions`
with assert statements for register length words ``__XWORD``

.. <legal notes>

legal notes
=================
| SPDX-FileCopyrightText: © 2022 ekvip automation GmbH <info@ekvip.de>
| SPDX-License-Identifier: Apache-2.0
| For details check: Apache-2.0_

.. _Apache-2.0: https://www.apache.org/licenses/LICENSE-2.0

.. </legal notes>

*)

PROPERTY x :IXwordAssertions
GET
x := THIS^.xwordAssertions;
END_GET
END_PROPERTY

END_FUNCTION_BLOCK

// ---- Assertor/Assertions/BitNumberAssertions/Word/classes/WordAssertions.TcPOU
(*

short summary
=================
This class provides assert statements for words  
It implements :ref:`IWordAssertions`

.. <legal notes>

legal notes
=================
| SPDX-FileCopyrightText: © 2022 ekvip automation GmbH <info@ekvip.de>
| SPDX-License-Identifier: Apache-2.0
| For details check: Apache-2.0_

.. _Apache-2.0: https://www.apache.org/licenses/LICENSE-2.0

.. </legal notes>

methods and properties
=======================

*)

{attribute 'reflection'}
FUNCTION_BLOCK INTERNAL WordAssertions EXTENDS AbstactAssertion IMPLEMENTS IWordAssertions
VAR
END_VAR
VAR CONSTANT
	(* least significant bit *)
	LSB	:WORD := 16#0001;
	(* most significant bit *)
	MSB :WORD := 16#8000;
END_VAR

(*

short summary
=================
This assertion method checks if the result current value bitwise ``AND`` mask is equal to the expected value

.. <legal notes>

legal notes
=================
| SPDX-FileCopyrightText: © 2022 ekvip automation GmbH <info@ekvip.de>
| SPDX-License-Identifier: Apache-2.0
| For details check: Apache-2.0_

.. _Apache-2.0: https://www.apache.org/licenses/LICENSE-2.0

.. </legal notes>

parameters
=================

*)

METHOD andMaskIsEqualTo
VAR_INPUT
	(* current value to check *)
	currentValue	:WORD;
	(* 2nd operand for bitwise operation *)
	mask			:WORD;
	(* expected result after masking *)
	expectedValue	:WORD;
	(* message if the assertion is false *)
	message			:AssertMessage;
END_VAR
IF ((currentValue AND mask) <> expectedValue) THEN
	THIS^.assertionWasWrong(message, THIS^.getDebugInfo('andMaskIsEqualTo'));
END_IF
END_METHOD

(*

short summary
=================
This assertion method checks if the result current value bitwise ``AND`` mask
is not equal to the unexpected value

.. <legal notes>

legal notes
=================
| SPDX-FileCopyrightText: © 2022 ekvip automation GmbH <info@ekvip.de>
| SPDX-License-Identifier: Apache-2.0
| For details check: Apache-2.0_

.. _Apache-2.0: https://www.apache.org/licenses/LICENSE-2.0

.. </legal notes>

parameters
=================

*)

METHOD andMaskIsNotEqualTo
VAR_INPUT
	(* current value to check *)
	currentValue	:WORD;
	(* 2nd operand for bitwise operation *)
	mask			:WORD;
	(* unexpected result after masking *)
	unexpectedValue	:WORD;
	(* message if the assertion is false *)
	message			:AssertMessage;
END_VAR
IF ((currentValue AND mask) = unexpectedValue) THEN
	THIS^.assertionWasWrong(message, THIS^.getDebugInfo('andMaskIsNotEqualTo'));
END_IF
END_METHOD

(*

short summary
=================
This assertion method checks if the selected bit of current value
is equal to the expected value

.. <legal notes>

legal notes
=================
| SPDX-FileCopyrightText: © 2022 ekvip automation GmbH <info@ekvip.de>
| SPDX-License-Identifier: Apache-2.0
| For details check: Apache-2.0_

.. _Apache-2.0: https://www.apache.org/licenses/LICENSE-2.0

.. </legal notes>

parameters
=================

*)

